LIN {X 0,Y 312.539,Z 409.82,A -85,B 0,C 180,E1 -15709.867,E2 -15709.867} C_VEL
LIN {X 0,Y 316.185,Z 420.984,A -85,B 0,C 180,E1 -15712.474,E2 -15712.474} C_VEL
LIN {X 0,Y 319.373,Z 431.927,A -85,B 0,C 180,E1 -15714.865,E2 -15714.865} C_VEL
LIN {X 0,Y 322.559,Z 445.519,A -85,B 0,C 180,E1 -15717.69,E2 -15717.69} C_VEL
LIN {X 0,Y 323.297,Z 449.924,A -85,B 0,C 180,E1 -15718.552,E2 -15718.552} C_VEL
LIN {X 0,Y 321.475,Z 469.515,A -85,B 0,C 180,E1 -15721.786,E2 -15721.786} C_VEL
LIN {X 0,Y 320.022,Z 488.05,A -85,B 0,C 180,E1 -15724.694,E2 -15724.694} C_VEL
LIN {X 0,Y 324.349,Z 518.766,A -85,B 0,C 180,E1 -15725.801,E2 -15725.801} C_VEL
LIN {X 0,Y 322.977,Z 585.301,A -85,B 0,C 180,E1 -15727.279,E2 -15727.279} C_VEL
LIN {X 0,Y 322.487,Z 602.467,A -85,B 0,C 180,E1 -15727.707,E2 -15727.707} C_VEL
LIN {X 0,Y 321.635,Z 615.557,A -85,B 0,C 180,E1 -15728.278,E2 -15728.278} C_VEL
LIN {X 0,Y 320.727,Z 627.617,A -85,B 0,C 180,E1 -15729.056,E2 -15729.056} C_VEL
LIN {X 0,Y 319.391,Z 639.348,A -85,B 0,C 180,E1 -15730.058,E2 -15730.058} C_VEL
LIN {X 0,Y 317.949,Z 650.541,A -85,B 0,C 180,E1 -15731.306,E2 -15731.306} C_VEL
LIN {X 0,Y 316.672,Z 660.214,A -85,B 0,C 180,E1 -15732.661,E2 -15732.661} C_VEL
LIN {X 0,Y 315.497,Z 668.968,A -85,B 0,C 180,E1 -15734.164,E2 -15734.164} C_VEL
LIN {X 0,Y 313.957,Z 677.978,A -85,B 0,C 180,E1 -15736.076,E2 -15736.076} C_VEL
LIN {X 0,Y 312.886,Z 685.206,A -85,B 0,C 180,E1 -15738.008,E2 -15738.008} C_VEL
LIN {X 0,Y 311.883,Z 691.838,A -85,B 0,C 180,E1 -15740.27,E2 -15740.27} C_VEL
LIN {X 0,Y 311.35,Z 696.194,A -85,B 0,C 180,E1 -15742.216,E2 -15742.216} C_VEL
LIN {X 0,Y 310.994,Z 699.108,A -85,B 0,C 180,E1 -15743.9,E2 -15743.9} C_VEL
LIN {X 0,Y 310.769,Z 701.783,A -85,B 0,C 180,E1 -15746.11,E2 -15746.11} C_VEL
LIN {X 0,Y 310.691,Z 702.783,A -85,B 0,C 180,E1 -15747.407,E2 -15747.407} C_VEL
LIN {X 0,Y 310.618,Z 703.635,A -85,B 0,C 180,E1 -15750,E2 -15750} C_VEL
LIN {X 0,Y 310.62,Z 703.44,A -85,B 0,C 180,E1 -15751.297,E2 -15751.297} C_VEL
LIN {X 0,Y 310.69,Z 702.849,A -85,B 0,C 180,E1 -15752.593,E2 -15752.593} C_VEL
LIN {X 0,Y 310.765,Z 701.874,A -85,B 0,C 180,E1 -15753.89,E2 -15753.89} C_VEL
LIN {X 0,Y 310.946,Z 699.383,A -85,B 0,C 180,E1 -15756.016,E2 -15756.016} C_VEL
LIN {X 0,Y 311.264,Z 696.397,A -85,B 0,C 180,E1 -15757.786,E2 -15757.786} C_VEL
LIN {X 0,Y 311.836,Z 692.102,A -85,B 0,C 180,E1 -15759.732,E2 -15759.732} C_VEL
LIN {X 0,Y 312.66,Z 686.615,A -85,B 0,C 180,E1 -15761.672,E2 -15761.672} C_VEL
LIN {X 0,Y 313.691,Z 679.736,A -85,B 0,C 180,E1 -15763.606,E2 -15763.606} C_VEL
LIN {X 0,Y 315.129,Z 671.132,A -85,B 0,C 180,E1 -15765.523,E2 -15765.523} C_VEL
LIN {X 0,Y 316.384,Z 662.938,A -85,B 0,C 180,E1 -15767.009,E2 -15767.009} C_VEL
LIN {X 0,Y 317.675,Z 652.616,A -85,B 0,C 180,E1 -15768.544,E2 -15768.544} C_VEL
LIN {X 0,Y 319.116,Z 641.878,A -85,B 0,C 180,E1 -15769.792,E2 -15769.792} C_VEL
LIN {X 0,Y 320.475,Z 629.948,A -85,B 0,C 180,E1 -15770.877,E2 -15770.877} C_VEL
LIN {X 0,Y 321.541,Z 617.429,A -85,B 0,C 180,E1 -15771.729,E2 -15771.729} C_VEL
LIN {X 0,Y 322.445,Z 604.145,A -85,B 0,C 180,E1 -15772.338,E2 -15772.338} C_VEL
LIN {X 0,Y 322.942,Z 589.97,A -85,B 0,C 180,E1 -15772.724,E2 -15772.724} C_VEL
LIN {X 0,Y 324.409,Z 518.731,A -85,B 0,C 180,E1 -15774.307,E2 -15774.307} C_VEL
LIN {X 0,Y 322.877,Z 507.001,A -85,B 0,C 180,E1 -15774.711,E2 -15774.711} C_VEL
LIN {X 0,Y 321.799,Z 503.315,A -85,B 0,C 180,E1 -15774.889,E2 -15774.889} C_VEL
LIN {X 0,Y 318.374,Z 497.993,A -85,B 0,C 180,E1 -15775.304,E2 -15775.304} C_VEL
LIN {X 0,Y 314.859,Z 492.705,A -85,B 0,C 180,E1 -15775.737,E2 -15775.737} C_VEL
LIN {X 0,Y 313.636,Z 489.058,A -85,B 0,C 180,E1 -15775.937,E2 -15775.937} C_VEL
LIN {X 0,Y 313.523,Z 487.144,A -85,B 0,C 180,E1 -15776.1,E2 -15776.1} C_VEL
LIN {X 0,Y 315.804,Z 461.684,A -85,B 0,C 180,E1 -15780.246,E2 -15780.246} C_VEL
LIN {X 0,Y 316.683,Z 451.244,A -85,B 0,C 180,E1 -15782.013,E2 -15782.013} C_VEL
LIN {X 0,Y 314.241,Z 439.793,A -85,B 0,C 180,E1 -15784.382,E2 -15784.382} C_VEL
LIN {X 0,Y 310.353,Z 425.27,A -85,B 0,C 180,E1 -15787.572,E2 -15787.572} C_VEL
LIN {X 0,Y 305.498,Z 410.99,A -85,B 0,C 180,E1 -15790.958,E2 -15790.958} C_VEL
LIN {X 0,Y 305.385,Z 410.45,A -85,B 0,C 180,E1 -15791.281,E2 -15791.281} C_VEL
LIN {X 0,Y 305.401,Z 410.414,A -85,B 0,C 180,E1 -15794.489,E2 -15794.489} C_VEL
LIN {X 0,Y 305.415,Z 410.443,A -85,B 0,C 180,E1 -15798.139,E2 -15798.139} C_VEL
LIN {X 0,Y 305.462,Z 410.432,A -85,B 0,C 180,E1 -15801.595,E2 -15801.595} C_VEL
LIN {X 0,Y 305.464,Z 410.436,A -85,B 0,C 180,E1 -15804.887,E2 -15804.887} C_VEL
LIN {X 0,Y 305.444,Z 410.439,A -85,B 0,C 180,E1 -15808.358,E2 -15808.358} C_VEL
LIN {X 0,Y 305.456,Z 410.422,A -85,B 0,C 180,E1 -15811.107,E2 -15811.107} C_VEL
LIN {X 0,Y 305.501,Z 410.431,A -85,B 0,C 180,E1 -15814.081,E2 -15814.081} C_VEL
LIN {X 0,Y 305.476,Z 410.417,A -85,B 0,C 180,E1 -15816.976,E2 -15816.976} C_VEL
LIN {X 0,Y 305.512,Z 410.414,A -85,B 0,C 180,E1 -15821.213,E2 -15821.213} C_VEL
LIN {X 0,Y 305.582,Z 410.421,A -85,B 0,C 180,E1 -15825.346,E2 -15825.346} C_VEL
LIN {X 0,Y 305.626,Z 410.392,A -85,B 0,C 180,E1 -15829.399,E2 -15829.399} C_VEL
LIN {X 0,Y 305.749,Z 410.399,A -85,B 0,C 180,E1 -15832.073,E2 -15832.073} C_VEL
LIN {X 0,Y 305.658,Z 410.387,A -85,B 0,C 180,E1 -15834.723,E2 -15834.723} C_VEL
LIN {X 0,Y 305.939,Z 410.374,A -85,B 0,C 180,E1 -15838.684,E2 -15838.684} C_VEL
LIN {X 0,Y 305.937,Z 410.356,A -85,B 0,C 180,E1 -15841.316,E2 -15841.316} C_VEL
LIN {X 0,Y 305.789,Z 410.393,A -85,B 0,C 180,E1 -15846.599,E2 -15846.599} C_VEL
LIN {X 0,Y 305.697,Z 410.381,A -85,B 0,C 180,E1 -15849.261,E2 -15849.261} C_VEL
LIN {X 0,Y 305.567,Z 410.422,A -85,B 0,C 180,E1 -15853.297,E2 -15853.297} C_VEL
LIN {X 0,Y 305.493,Z 410.407,A -85,B 0,C 180,E1 -15856.026,E2 -15856.026} C_VEL
LIN {X 0,Y 305.478,Z 410.433,A -85,B 0,C 180,E1 -15860.188,E2 -15860.188} C_VEL
LIN {X 0,Y 305.443,Z 410.425,A -85,B 0,C 180,E1 -15864.467,E2 -15864.467} C_VEL
LIN {X 0,Y 305.444,Z 410.431,A -85,B 0,C 180,E1 -15867.399,E2 -15867.399} C_VEL
LIN {X 0,Y 305.419,Z 410.43,A -85,B 0,C 180,E1 -15870.414,E2 -15870.414} C_VEL
LIN {X 0,Y 305.466,Z 410.419,A -85,B 0,C 180,E1 -15874.078,E2 -15874.078} C_VEL
LIN {X 0,Y 305.453,Z 410.437,A -85,B 0,C 180,E1 -15876.743,E2 -15876.743} C_VEL
LIN {X 0,Y 305.41,Z 410.388,A -85,B 0,C 180,E1 -15880.589,E2 -15880.589} C_VEL
LIN {X 0,Y 305.422,Z 410.412,A -85,B 0,C 180,E1 -15883.656,E2 -15883.656} C_VEL
LIN {X 0,Y 305.435,Z 410.407,A -85,B 0,C 180,E1 -15887.418,E2 -15887.418} C_VEL
LIN {X 0,Y 305.448,Z 410.435,A -85,B 0,C 180,E1 -15891.593,E2 -15891.593} C_VEL
LIN {X 0,Y 305.529,Z 410.634,A -85,B 0,C 180,E1 -15893.411,E2 -15893.411} C_VEL
LIN {X 0,Y 308.682,Z 425.243,A -85,B 0,C 180,E1 -15896.877,E2 -15896.877} C_VEL
LIN {X 0,Y 311.225,Z 437.046,A -85,B 0,C 180,E1 -15899.561,E2 -15899.561} C_VEL
LIN {X 0,Y 311.159,Z 440.07,A -85,B 0,C 180,E1 -15900.204,E2 -15900.204} C_VEL
LIN {X 0,Y 311.02,Z 441.837,A -85,B 0,C 180,E1 -15900.497,E2 -15900.497} C_VEL
LIN {X 0,Y 312.83,Z 473.685,A -85,B 0,C 180,E1 -15903.011,E2 -15903.011} C_VEL
LIN {X 0,Y 313.362,Z 488.832,A -85,B 0,C 180,E1 -15904.212,E2 -15904.212} C_VEL
LIN {X 0,Y 316.809,Z 520.766,A -85,B 0,C 180,E1 -15905.295,E2 -15905.295} C_VEL
LIN {X 0,Y 317.335,Z 528.316,A -85,B 0,C 180,E1 -15905.522,E2 -15905.522} C_VEL
LIN {X 0,Y 315.578,Z 604.063,A -85,B 0,C 180,E1 -15907.235,E2 -15907.235} C_VEL
LIN {X 0,Y 314.795,Z 617.344,A -85,B 0,C 180,E1 -15907.738,E2 -15907.738} C_VEL
LIN {X 0,Y 313.773,Z 629.822,A -85,B 0,C 180,E1 -15908.483,E2 -15908.483} C_VEL
LIN {X 0,Y 312.624,Z 641.462,A -85,B 0,C 180,E1 -15909.435,E2 -15909.435} C_VEL
LIN {X 0,Y 311.242,Z 652.056,A -85,B 0,C 180,E1 -15910.545,E2 -15910.545} C_VEL
LIN {X 0,Y 309.74,Z 662.85,A -85,B 0,C 180,E1 -15911.992,E2 -15911.992} C_VEL
LIN {X 0,Y 308.35,Z 672.278,A -85,B 0,C 180,E1 -15913.57,E2 -15913.57} C_VEL
LIN {X 0,Y 307.006,Z 681.154,A -85,B 0,C 180,E1 -15915.415,E2 -15915.415} C_VEL
LIN {X 0,Y 305.735,Z 688.702,A -85,B 0,C 180,E1 -15917.386,E2 -15917.386} C_VEL
LIN {X 0,Y 304.903,Z 694.761,A -85,B 0,C 180,E1 -15919.374,E2 -15919.374} C_VEL
LIN {X 0,Y 304.256,Z 699.543,A -85,B 0,C 180,E1 -15921.365,E2 -15921.365} C_VEL
LIN {X 0,Y 303.913,Z 703.193,A -85,B 0,C 180,E1 -15923.36,E2 -15923.36} C_VEL
LIN {X 0,Y 303.761,Z 705.073,A -85,B 0,C 180,E1 -15924.69,E2 -15924.69} C_VEL
LIN {X 0,Y 303.702,Z 706.49,A -85,B 0,C 180,E1 -15926.019,E2 -15926.019} C_VEL
LIN {X 0,Y 303.658,Z 707.49,A -85,B 0,C 180,E1 -15927.347,E2 -15927.347} C_VEL
LIN {X 0,Y 303.597,Z 708.1,A -85,B 0,C 180,E1 -15928.673,E2 -15928.673} C_VEL
LIN {X 0,Y 303.616,Z 708.317,A -85,B 0,C 180,E1 -15930,E2 -15930} C_VEL
LIN {X 0,Y 303.626,Z 708.094,A -85,B 0,C 180,E1 -15931.326,E2 -15931.326} C_VEL
LIN {X 0,Y 303.665,Z 707.479,A -85,B 0,C 180,E1 -15932.653,E2 -15932.653} C_VEL
LIN {X 0,Y 303.723,Z 706.475,A -85,B 0,C 180,E1 -15933.98,E2 -15933.98} C_VEL
LIN {X 0,Y 303.825,Z 704.233,A -85,B 0,C 180,E1 -15935.92,E2 -15935.92} C_VEL
LIN {X 0,Y 304.103,Z 700.848,A -85,B 0,C 180,E1 -15937.97,E2 -15937.97} C_VEL
LIN {X 0,Y 304.692,Z 696.451,A -85,B 0,C 180,E1 -15939.962,E2 -15939.962} C_VEL
LIN {X 0,Y 305.604,Z 689.751,A -85,B 0,C 180,E1 -15942.282,E2 -15942.282} C_VEL
LIN {X 0,Y 306.777,Z 682.429,A -85,B 0,C 180,E1 -15944.257,E2 -15944.257} C_VEL
LIN {X 0,Y 308.121,Z 673.606,A -85,B 0,C 180,E1 -15946.163,E2 -15946.163} C_VEL
LIN {X 0,Y 309.554,Z 663.768,A -85,B 0,C 180,E1 -15947.848,E2 -15947.848} C_VEL
LIN {X 0,Y 311.059,Z 653.202,A -85,B 0,C 180,E1 -15949.295,E2 -15949.295} C_VEL
LIN {X 0,Y 312.382,Z 642.956,A -85,B 0,C 180,E1 -15950.409,E2 -15950.409} C_VEL
LIN {X 0,Y 313.685,Z 630.643,A -85,B 0,C 180,E1 -15951.437,E2 -15951.437} C_VEL
LIN {X 0,Y 314.762,Z 618.361,A -85,B 0,C 180,E1 -15952.221,E2 -15952.221} C_VEL
LIN {X 0,Y 317.898,Z 604.839,A -85,B 0,C 180,E1 -15953.622,E2 -15953.622} C_VEL
LIN {X 0,Y 320.563,Z 591.482,A -85,B 0,C 180,E1 -15954.704,E2 -15954.704} C_VEL
LIN {X 0,Y 322.77,Z 577.813,A -85,B 0,C 180,E1 -15955.556,E2 -15955.556} C_VEL
LIN {X 0,Y 324.493,Z 563.284,A -85,B 0,C 180,E1 -15956.229,E2 -15956.229} C_VEL
LIN {X 0,Y 327.437,Z 528.631,A -85,B 0,C 180,E1 -15957.532,E2 -15957.532} C_VEL
LIN {X 0,Y 327.503,Z 512.069,A -85,B 0,C 180,E1 -15958.423,E2 -15958.423} C_VEL
LIN {X 0,Y 326.752,Z 496.351,A -85,B 0,C 180,E1 -15959.479,E2 -15959.479} C_VEL
LIN {X 0,Y 325.256,Z 480.762,A -85,B 0,C 180,E1 -15960.768,E2 -15960.768} C_VEL
LIN {X 0,Y 323.384,Z 466.341,A -85,B 0,C 180,E1 -15962.201,E2 -15962.201} C_VEL
LIN {X 0,Y 322.036,Z 457.299,A -85,B 0,C 180,E1 -15963.249,E2 -15963.249} C_VEL
LIN {X 0,Y 319.695,Z 451.276,A -85,B 0,C 180,E1 -15964.432,E2 -15964.432} C_VEL
LIN {X 0,Y 315.876,Z 442.522,A -85,B 0,C 180,E1 -15966.702,E2 -15966.702} C_VEL
LIN {X 0,Y 314.394,Z 436.999,A -85,B 0,C 180,E1 -15969.172,E2 -15969.172} C_VEL
LIN {X 0,Y 313.453,Z 433.635,A -85,B 0,C 180,E1 -15970.993,E2 -15970.993} C_VEL
LIN {X 0,Y 312.007,Z 429.364,A -85,B 0,C 180,E1 -15973.879,E2 -15973.879} C_VEL
LIN {X 0,Y 310.757,Z 425.66,A -85,B 0,C 180,E1 -15977.276,E2 -15977.276} C_VEL
LIN {X 0,Y 310.242,Z 424.091,A -85,B 0,C 180,E1 -15979.629,E2 -15979.629} C_VEL
LIN {X 0,Y 311.764,Z 424.945,A -85,B 0,C 180,E1 -15981.669,E2 -15981.669} C_VEL
LIN {X 0,Y 313.944,Z 425.846,A -85,B 0,C 180,E1 -15983.379,E2 -15983.379} C_VEL
LIN {X 0,Y 316.792,Z 428.045,A -85,B 0,C 180,E1 -15985.169,E2 -15985.169} C_VEL
LIN {X 0,Y 320.809,Z 431.911,A -85,B 0,C 180,E1 -15987.214,E2 -15987.214} C_VEL
LIN {X 0,Y 323.364,Z 434.77,A -85,B 0,C 180,E1 -15988.331,E2 -15988.331} C_VEL
LIN {X 0,Y 324.917,Z 437.076,A -85,B 0,C 180,E1 -15989,E2 -15989} C_VEL
LIN {X 0,Y 329.004,Z 443.809,A -85,B 0,C 180,E1 -15990.619,E2 -15990.619} C_VEL
LIN {X 0,Y 333.23,Z 452.024,A -85,B 0,C 180,E1 -15992.145,E2 -15992.145} C_VEL
LIN {X 0,Y 329.446,Z 489.733,A -85,B 0,C 180,E1 -15993.634,E2 -15993.634} C_VEL
LIN {X 0,Y 328.128,Z 509.636,A -85,B 0,C 180,E1 -15994.552,E2 -15994.552} C_VEL
LIN {X 0,Y 326.845,Z 523.763,A -85,B 0,C 180,E1 -15995.472,E2 -15995.472} C_VEL
LIN {X 0,Y 325.453,Z 535.265,A -85,B 0,C 180,E1 -15996.453,E2 -15996.453} C_VEL
LIN {X 0,Y 323.679,Z 546.599,A -85,B 0,C 180,E1 -15997.668,E2 -15997.668} C_VEL
LIN {X 0,Y 321.413,Z 557.833,A -85,B 0,C 180,E1 -15999.187,E2 -15999.187} C_VEL
LIN {X 0,Y 319.436,Z 566.96,A -85,B 0,C 180,E1 -16000.73,E2 -16000.73} C_VEL
LIN {X 0,Y 317.213,Z 575.546,A -85,B 0,C 180,E1 -16002.534,E2 -16002.534} C_VEL
LIN {X 0,Y 315.008,Z 582.876,A -85,B 0,C 180,E1 -16004.471,E2 -16004.471} C_VEL
LIN {X 0,Y 313.158,Z 588.479,A -85,B 0,C 180,E1 -16006.37,E2 -16006.37} C_VEL
LIN {X 0,Y 311.44,Z 592.85,A -85,B 0,C 180,E1 -16008.282,E2 -16008.282} C_VEL
LIN {X 0,Y 310.478,Z 595.11,A -85,B 0,C 180,E1 -16009.567,E2 -16009.567} C_VEL
LIN {X 0,Y 309.561,Z 596.914,A -85,B 0,C 180,E1 -16010.856,E2 -16010.856} C_VEL
LIN {X 0,Y 308.695,Z 598.235,A -85,B 0,C 180,E1 -16012.149,E2 -16012.149} C_VEL
LIN {X 0,Y 308.072,Z 599.122,A -85,B 0,C 180,E1 -16013.45,E2 -16013.45} C_VEL
LIN {X 0,Y 307.598,Z 599.575,A -85,B 0,C 180,E1 -16014.756,E2 -16014.756} C_VEL
LIN {X 0,Y 307.124,Z 599.575,A -85,B 0,C 180,E1 -16016.064,E2 -16016.064} C_VEL
LIN {X 0,Y 306.617,Z 599.175,A -85,B 0,C 180,E1 -16017.373,E2 -16017.373} C_VEL
LIN {X 0,Y 306.293,Z 598.342,A -85,B 0,C 180,E1 -16018.685,E2 -16018.685} C_VEL
LIN {X 0,Y 305.867,Z 597.074,A -85,B 0,C 180,E1 -16020,E2 -16020} C_VEL
LIN {X 0,Y 305.752,Z 594.31,A -85,B 0,C 180,E1 -16021.976,E2 -16021.976} C_VEL
LIN {X 0,Y 305.613,Z 590.502,A -85,B 0,C 180,E1 -16023.956,E2 -16023.956} C_VEL
LIN {X 0,Y 305.81,Z 585.528,A -85,B 0,C 180,E1 -16025.936,E2 -16025.936} C_VEL
LIN {X 0,Y 306.111,Z 579.272,A -85,B 0,C 180,E1 -16027.918,E2 -16027.918} C_VEL
LIN {X 0,Y 306.582,Z 571.477,A -85,B 0,C 180,E1 -16029.914,E2 -16029.914} C_VEL
LIN {X 0,Y 307.077,Z 561.898,A -85,B 0,C 180,E1 -16031.887,E2 -16031.887} C_VEL
LIN {X 0,Y 307.669,Z 552.084,A -85,B 0,C 180,E1 -16033.541,E2 -16033.541} C_VEL
LIN {X 0,Y 308.288,Z 541.233,A -85,B 0,C 180,E1 -16035.029,E2 -16035.029} C_VEL
LIN {X 0,Y 308.947,Z 529.369,A -85,B 0,C 180,E1 -16036.35,E2 -16036.35} C_VEL
LIN {X 0,Y 309.453,Z 516.504,A -85,B 0,C 180,E1 -16037.471,E2 -16037.471} C_VEL
LIN {X 0,Y 309.903,Z 503.178,A -85,B 0,C 180,E1 -16038.352,E2 -16038.352} C_VEL
LIN {X 0,Y 310.218,Z 488.806,A -85,B 0,C 180,E1 -16039.006,E2 -16039.006} C_VEL
LIN {X 0,Y 311.04,Z 448.886,A -85,B 0,C 180,E1 -16040.32,E2 -16040.32} C_VEL
LIN {X 0,Y 311.496,Z 430.443,A -85,B 0,C 180,E1 -16040.934,E2 -16040.934} C_VEL
LIN {X 0,Y 305.728,Z 411.446,A -85,B 0,C 180,E1 -16041.846,E2 -16041.846} C_VEL
LIN {X 0,Y 305.565,Z 410.535,A -85,B 0,C 180,E1 -16042.08,E2 -16042.08} C_VEL
LIN {X 0,Y 305.475,Z 410.434,A -85,B 0,C 180,E1 -16046.199,E2 -16046.199} C_VEL
LIN {X 0,Y 305.46,Z 410.416,A -85,B 0,C 180,E1 -16049.037,E2 -16049.037} C_VEL
LIN {X 0,Y 305.438,Z 410.439,A -85,B 0,C 180,E1 -16051.953,E2 -16051.953} C_VEL
LIN {X 0,Y 305.464,Z 410.426,A -85,B 0,C 180,E1 -16055.113,E2 -16055.113} C_VEL
LIN {X 0,Y 305.442,Z 410.426,A -85,B 0,C 180,E1 -16058.527,E2 -16058.527} C_VEL
LIN {X 0,Y 305.456,Z 410.428,A -85,B 0,C 180,E1 -16062.586,E2 -16062.586} C_VEL
LIN {X 0,Y 305.427,Z 410.438,A -85,B 0,C 180,E1 -16066.345,E2 -16066.345} C_VEL
LIN {X 0,Y 305.476,Z 410.634,A -85,B 0,C 180,E1 -16069.052,E2 -16069.052} C_VEL
LIN {X 0,Y 309.593,Z 423.12,A -85,B 0,C 180,E1 -16072.086,E2 -16072.086} C_VEL
LIN {X 0,Y 312.806,Z 434.138,A -85,B 0,C 180,E1 -16074.532,E2 -16074.532} C_VEL
LIN {X 0,Y 316.219,Z 448.825,A -85,B 0,C 180,E1 -16077.625,E2 -16077.625} C_VEL
LIN {X 0,Y 316.664,Z 452.335,A -85,B 0,C 180,E1 -16078.302,E2 -16078.302} C_VEL
LIN {X 0,Y 314.685,Z 472.51,A -85,B 0,C 180,E1 -16081.668,E2 -16081.668} C_VEL
LIN {X 0,Y 313.435,Z 487.99,A -85,B 0,C 180,E1 -16084.12,E2 -16084.12} C_VEL
LIN {X 0,Y 317.883,Z 519.622,A -85,B 0,C 180,E1 -16085.298,E2 -16085.298} C_VEL
LIN {X 0,Y 316.456,Z 585.266,A -85,B 0,C 180,E1 -16086.784,E2 -16086.784} C_VEL
LIN {X 0,Y 315.946,Z 602.471,A -85,B 0,C 180,E1 -16087.22,E2 -16087.22} C_VEL
LIN {X 0,Y 315.06,Z 615.582,A -85,B 0,C 180,E1 -16087.801,E2 -16087.801} C_VEL
LIN {X 0,Y 314.116,Z 627.654,A -85,B 0,C 180,E1 -16088.594,E2 -16088.594} C_VEL
LIN {X 0,Y 312.737,Z 639.391,A -85,B 0,C 180,E1 -16089.615,E2 -16089.615} C_VEL
LIN {X 0,Y 311.233,Z 650.587,A -85,B 0,C 180,E1 -16090.887,E2 -16090.887} C_VEL
LIN {X 0,Y 309.698,Z 661.567,A -85,B 0,C 180,E1 -16092.473,E2 -16092.473} C_VEL
LIN {X 0,Y 308.342,Z 670.653,A -85,B 0,C 180,E1 -16094.127,E2 -16094.127} C_VEL
LIN {X 0,Y 306.834,Z 679.356,A -85,B 0,C 180,E1 -16096.084,E2 -16096.084} C_VEL
LIN {X 0,Y 305.743,Z 686.341,A -85,B 0,C 180,E1 -16098.061,E2 -16098.061} C_VEL
LIN {X 0,Y 304.861,Z 691.892,A -85,B 0,C 180,E1 -16100.044,E2 -16100.044} C_VEL
LIN {X 0,Y 304.294,Z 696.248,A -85,B 0,C 180,E1 -16102.035,E2 -16102.035} C_VEL
LIN {X 0,Y 303.886,Z 699.461,A -85,B 0,C 180,E1 -16103.971,E2 -16103.971} C_VEL
LIN {X 0,Y 303.687,Z 701.837,A -85,B 0,C 180,E1 -16106.019,E2 -16106.019} C_VEL
LIN {X 0,Y 303.617,Z 702.837,A -85,B 0,C 180,E1 -16107.347,E2 -16107.347} C_VEL
LIN {X 0,Y 303.535,Z 703.689,A -85,B 0,C 180,E1 -16110,E2 -16110} C_VEL
LIN {X 0,Y 303.539,Z 703.493,A -85,B 0,C 180,E1 -16111.327,E2 -16111.327} C_VEL
LIN {X 0,Y 303.617,Z 702.902,A -85,B 0,C 180,E1 -16112.654,E2 -16112.654} C_VEL
LIN {X 0,Y 303.683,Z 701.928,A -85,B 0,C 180,E1 -16113.981,E2 -16113.981} C_VEL
LIN {X 0,Y 303.872,Z 699.638,A -85,B 0,C 180,E1 -16116.004,E2 -16116.004} C_VEL
LIN {X 0,Y 304.231,Z 696.449,A -85,B 0,C 180,E1 -16117.967,E2 -16117.967} C_VEL
LIN {X 0,Y 304.817,Z 692.153,A -85,B 0,C 180,E1 -16119.958,E2 -16119.958} C_VEL
LIN {X 0,Y 305.694,Z 686.665,A -85,B 0,C 180,E1 -16121.942,E2 -16121.942} C_VEL
LIN {X 0,Y 306.78,Z 679.784,A -85,B 0,C 180,E1 -16123.919,E2 -16123.919} C_VEL
LIN {X 0,Y 308.281,Z 671.178,A -85,B 0,C 180,E1 -16125.877,E2 -16125.877} C_VEL
LIN {X 0,Y 309.668,Z 661.826,A -85,B 0,C 180,E1 -16127.597,E2 -16127.597} C_VEL
LIN {X 0,Y 311.131,Z 651.407,A -85,B 0,C 180,E1 -16129.119,E2 -16129.119} C_VEL
LIN {X 0,Y 312.649,Z 640.386,A -85,B 0,C 180,E1 -16130.391,E2 -16130.391} C_VEL
LIN {X 0,Y 313.853,Z 629.974,A -85,B 0,C 180,E1 -16131.339,E2 -16131.339} C_VEL
LIN {X 0,Y 314.972,Z 617.437,A -85,B 0,C 180,E1 -16132.206,E2 -16132.206} C_VEL
LIN {X 0,Y 315.899,Z 604.125,A -85,B 0,C 180,E1 -16132.827,E2 -16132.827} C_VEL
LIN {X 0,Y 316.419,Z 589.888,A -85,B 0,C 180,E1 -16133.219,E2 -16133.219} C_VEL
LIN {X 0,Y 317.94,Z 519.507,A -85,B 0,C 180,E1 -16134.813,E2 -16134.813} C_VEL
LIN {X 0,Y 313.636,Z 489.058,A -85,B 0,C 180,E1 -16135.937,E2 -16135.937} C_VEL
LIN {X 0,Y 312.94,Z 486.827,A -85,B 0,C 180,E1 -16136.204,E2 -16136.204} C_VEL
LIN {X 0,Y 310.285,Z 479.752,A -85,B 0,C 180,E1 -16137.628,E2 -16137.628} C_VEL
LIN {X 0,Y 308.746,Z 472.042,A -85,B 0,C 180,E1 -16139.145,E2 -16139.145} C_VEL
LIN {X 0,Y 308.815,Z 467.004,A -85,B 0,C 180,E1 -16140.001,E2 -16140.001} C_VEL
LIN {X 0,Y 310.097,Z 454.673,A -85,B 0,C 180,E1 -16142.095,E2 -16142.095} C_VEL
LIN {X 0,Y 309.637,Z 450.645,A -85,B 0,C 180,E1 -16142.88,E2 -16142.88} C_VEL
LIN {X 0,Y 306.672,Z 438.007,A -85,B 0,C 180,E1 -16145.596,E2 -16145.596} C_VEL
LIN {X 0,Y 303.141,Z 425.405,A -85,B 0,C 180,E1 -16148.467,E2 -16148.467} C_VEL
LIN {X 0,Y 298.41,Z 411.555,A -85,B 0,C 180,E1 -16151.906,E2 -16151.906} C_VEL
LIN {X 0,Y 298.373,Z 411.305,A -85,B 0,C 180,E1 -16153.098,E2 -16153.098} C_VEL
LIN {X 0,Y 298.373,Z 411.313,A -85,B 0,C 180,E1 -16156.915,E2 -16156.915} C_VEL
LIN {X 0,Y 298.387,Z 411.32,A -85,B 0,C 180,E1 -16161.011,E2 -16161.011} C_VEL
LIN {X 0,Y 298.407,Z 411.311,A -85,B 0,C 180,E1 -16163.928,E2 -16163.928} C_VEL
LIN {X 0,Y 298.395,Z 411.303,A -85,B 0,C 180,E1 -16167.2,E2 -16167.2} C_VEL
LIN {X 0,Y 298.367,Z 411.306,A -85,B 0,C 180,E1 -16170.638,E2 -16170.638} C_VEL
LIN {X 0,Y 298.441,Z 411.304,A -85,B 0,C 180,E1 -16174.92,E2 -16174.92} C_VEL
LIN {X 0,Y 298.402,Z 411.306,A -85,B 0,C 180,E1 -16177.862,E2 -16177.862} C_VEL
LIN {X 0,Y 298.463,Z 411.298,A -85,B 0,C 180,E1 -16180.752,E2 -16180.752} C_VEL
LIN {X 0,Y 298.514,Z 411.3,A -85,B 0,C 180,E1 -16184.991,E2 -16184.991} C_VEL
LIN {X 0,Y 298.584,Z 411.267,A -85,B 0,C 180,E1 -16189.146,E2 -16189.146} C_VEL
LIN {X 0,Y 298.701,Z 411.279,A -85,B 0,C 180,E1 -16191.884,E2 -16191.884} C_VEL
LIN {X 0,Y 298.628,Z 411.263,A -85,B 0,C 180,E1 -16194.598,E2 -16194.598} C_VEL
LIN {X 0,Y 298.907,Z 411.25,A -85,B 0,C 180,E1 -16198.653,E2 -16198.653} C_VEL
LIN {X 0,Y 298.905,Z 411.23,A -85,B 0,C 180,E1 -16201.347,E2 -16201.347} C_VEL
LIN {X 0,Y 298.738,Z 411.271,A -85,B 0,C 180,E1 -16206.755,E2 -16206.755} C_VEL
LIN {X 0,Y 298.628,Z 411.26,A -85,B 0,C 180,E1 -16209.482,E2 -16209.482} C_VEL
LIN {X 0,Y 298.518,Z 411.301,A -85,B 0,C 180,E1 -16213.617,E2 -16213.617} C_VEL
LIN {X 0,Y 298.43,Z 411.284,A -85,B 0,C 180,E1 -16216.415,E2 -16216.415} C_VEL
LIN {X 0,Y 298.433,Z 411.311,A -85,B 0,C 180,E1 -16219.611,E2 -16219.611} C_VEL
LIN {X 0,Y 298.384,Z 411.294,A -85,B 0,C 180,E1 -16223.604,E2 -16223.604} C_VEL
LIN {X 0,Y 298.403,Z 411.313,A -85,B 0,C 180,E1 -16226.583,E2 -16226.583} C_VEL
LIN {X 0,Y 298.359,Z 411.301,A -85,B 0,C 180,E1 -16229.648,E2 -16229.648} C_VEL
LIN {X 0,Y 298.395,Z 411.313,A -85,B 0,C 180,E1 -16232.8,E2 -16232.8} C_VEL
LIN {X 0,Y 298.405,Z 411.31,A -85,B 0,C 180,E1 -16236.072,E2 -16236.072} C_VEL
LIN {X 0,Y 298.375,Z 411.279,A -85,B 0,C 180,E1 -16239.492,E2 -16239.492} C_VEL
LIN {X 0,Y 298.37,Z 411.276,A -85,B 0,C 180,E1 -16243.097,E2 -16243.097} C_VEL
LIN {X 0,Y 298.371,Z 411.296,A -85,B 0,C 180,E1 -16246.914,E2 -16246.914} C_VEL
LIN {X 0,Y 298.356,Z 411.301,A -85,B 0,C 180,E1 -16251.018,E2 -16251.018} C_VEL
LIN {X 0,Y 298.497,Z 411.542,A -85,B 0,C 180,E1 -16253.18,E2 -16253.18} C_VEL
LIN {X 0,Y 301.836,Z 427.164,A -85,B 0,C 180,E1 -16256.954,E2 -16256.954} C_VEL
LIN {X 0,Y 304.14,Z 437.746,A -85,B 0,C 180,E1 -16259.365,E2 -16259.365} C_VEL
LIN {X 0,Y 304.859,Z 443.301,A -85,B 0,C 180,E1 -16259.907,E2 -16259.907} C_VEL
LIN {X 0,Y 306.463,Z 474.151,A -85,B 0,C 180,E1 -16262.416,E2 -16262.416} C_VEL
LIN {X 0,Y 306.86,Z 488.84,A -85,B 0,C 180,E1 -16263.622,E2 -16263.622} C_VEL
LIN {X 0,Y 310.309,Z 520.688,A -85,B 0,C 180,E1 -16264.738,E2 -16264.738} C_VEL
LIN {X 0,Y 310.859,Z 529.725,A -85,B 0,C 180,E1 -16265.01,E2 -16265.01} C_VEL
LIN {X 0,Y 309.063,Z 604.111,A -85,B 0,C 180,E1 -16266.727,E2 -16266.727} C_VEL
LIN {X 0,Y 308.275,Z 616.535,A -85,B 0,C 180,E1 -16267.197,E2 -16267.197} C_VEL
LIN {X 0,Y 307.286,Z 628.691,A -85,B 0,C 180,E1 -16267.917,E2 -16267.917} C_VEL
LIN {X 0,Y 305.995,Z 641.431,A -85,B 0,C 180,E1 -16268.969,E2 -16268.969} C_VEL
LIN {X 0,Y 304.567,Z 652.019,A -85,B 0,C 180,E1 -16270.101,E2 -16270.101} C_VEL
LIN {X 0,Y 302.967,Z 662.807,A -85,B 0,C 180,E1 -16271.575,E2 -16271.575} C_VEL
LIN {X 0,Y 301.485,Z 672.554,A -85,B 0,C 180,E1 -16273.249,E2 -16273.249} C_VEL
LIN {X 0,Y 300.133,Z 681.106,A -85,B 0,C 180,E1 -16275.073,E2 -16275.073} C_VEL
LIN {X 0,Y 298.794,Z 688.652,A -85,B 0,C 180,E1 -16277.088,E2 -16277.088} C_VEL
LIN {X 0,Y 297.885,Z 694.71,A -85,B 0,C 180,E1 -16279.12,E2 -16279.12} C_VEL
LIN {X 0,Y 297.217,Z 699.491,A -85,B 0,C 180,E1 -16281.158,E2 -16281.158} C_VEL
LIN {X 0,Y 296.846,Z 703.14,A -85,B 0,C 180,E1 -16283.201,E2 -16283.201} C_VEL
LIN {X 0,Y 296.689,Z 705.02,A -85,B 0,C 180,E1 -16284.563,E2 -16284.563} C_VEL
LIN {X 0,Y 296.601,Z 706.437,A -85,B 0,C 180,E1 -16285.923,E2 -16285.923} C_VEL
LIN {X 0,Y 296.584,Z 707.437,A -85,B 0,C 180,E1 -16287.283,E2 -16287.283} C_VEL
LIN {X 0,Y 296.516,Z 708.047,A -85,B 0,C 180,E1 -16288.642,E2 -16288.642} C_VEL
LIN {X 0,Y 296.53,Z 708.263,A -85,B 0,C 180,E1 -16290,E2 -16290} C_VEL
LIN {X 0,Y 296.544,Z 708.04,A -85,B 0,C 180,E1 -16291.358,E2 -16291.358} C_VEL
LIN {X 0,Y 296.59,Z 707.425,A -85,B 0,C 180,E1 -16292.716,E2 -16292.716} C_VEL
LIN {X 0,Y 296.639,Z 706.421,A -85,B 0,C 180,E1 -16294.076,E2 -16294.076} C_VEL
LIN {X 0,Y 296.738,Z 704.415,A -85,B 0,C 180,E1 -16295.88,E2 -16295.88} C_VEL
LIN {X 0,Y 297.061,Z 700.794,A -85,B 0,C 180,E1 -16298.161,E2 -16298.161} C_VEL
LIN {X 0,Y 297.66,Z 696.397,A -85,B 0,C 180,E1 -16300.2,E2 -16300.2} C_VEL
LIN {X 0,Y 298.625,Z 689.697,A -85,B 0,C 180,E1 -16302.574,E2 -16302.574} C_VEL
LIN {X 0,Y 299.869,Z 682.377,A -85,B 0,C 180,E1 -16304.593,E2 -16304.593} C_VEL
LIN {X 0,Y 301.266,Z 673.71,A -85,B 0,C 180,E1 -16306.51,E2 -16306.51} C_VEL
LIN {X 0,Y 302.792,Z 663.719,A -85,B 0,C 180,E1 -16308.261,E2 -16308.261} C_VEL
LIN {X 0,Y 304.375,Z 653.156,A -85,B 0,C 180,E1 -16309.736,E2 -16309.736} C_VEL
LIN {X 0,Y 305.728,Z 642.914,A -85,B 0,C 180,E1 -16310.874,E2 -16310.874} C_VEL
LIN {X 0,Y 307.095,Z 630.609,A -85,B 0,C 180,E1 -16311.92,E2 -16311.92} C_VEL
LIN {X 0,Y 307.982,Z 620.933,A -85,B 0,C 180,E1 -16312.56,E2 -16312.56} C_VEL
LIN {X 0,Y 311.125,Z 608.476,A -85,B 0,C 180,E1 -16313.991,E2 -16313.991} C_VEL
LIN {X 0,Y 314.052,Z 595.572,A -85,B 0,C 180,E1 -16315.163,E2 -16315.163} C_VEL
LIN {X 0,Y 316.719,Z 581.3,A -85,B 0,C 180,E1 -16316.169,E2 -16316.169} C_VEL
LIN {X 0,Y 318.938,Z 566.333,A -85,B 0,C 180,E1 -16316.943,E2 -16316.943} C_VEL
LIN {X 0,Y 322.373,Z 529.81,A -85,B 0,C 180,E1 -16318.378,E2 -16318.378} C_VEL
LIN {X 0,Y 322.579,Z 513.411,A -85,B 0,C 180,E1 -16319.298,E2 -16319.298} C_VEL
LIN {X 0,Y 322.034,Z 498.47,A -85,B 0,C 180,E1 -16320.345,E2 -16320.345} C_VEL
LIN {X 0,Y 320.86,Z 483.7,A -85,B 0,C 180,E1 -16321.608,E2 -16321.608} C_VEL
LIN {X 0,Y 319.33,Z 469.773,A -85,B 0,C 180,E1 -16323.037,E2 -16323.037} C_VEL
LIN {X 0,Y 318.265,Z 461.755,A -85,B 0,C 180,E1 -16323.994,E2 -16323.994} C_VEL
LIN {X 0,Y 316.441,Z 456.645,A -85,B 0,C 180,E1 -16325.045,E2 -16325.045} C_VEL
LIN {X 0,Y 312.699,Z 447.681,A -85,B 0,C 180,E1 -16327.447,E2 -16327.447} C_VEL
LIN {X 0,Y 309.214,Z 440.368,A -85,B 0,C 180,E1 -16330.353,E2 -16330.353} C_VEL
LIN {X 0,Y 307.507,Z 435.89,A -85,B 0,C 180,E1 -16332.862,E2 -16332.862} C_VEL
LIN {X 0,Y 306.833,Z 433.197,A -85,B 0,C 180,E1 -16335.239,E2 -16335.239} C_VEL
LIN {X 0,Y 307.058,Z 431.726,A -85,B 0,C 180,E1 -16337.332,E2 -16337.332} C_VEL
LIN {X 0,Y 307.757,Z 431.059,A -85,B 0,C 180,E1 -16338.903,E2 -16338.903} C_VEL
LIN {X 0,Y 309.708,Z 431.684,A -85,B 0,C 180,E1 -16341.415,E2 -16341.415} C_VEL
LIN {X 0,Y 311.962,Z 432.588,A -85,B 0,C 180,E1 -16343.231,E2 -16343.231} C_VEL
LIN {X 0,Y 314.638,Z 434.745,A -85,B 0,C 180,E1 -16344.971,E2 -16344.971} C_VEL
LIN {X 0,Y 318.216,Z 438.206,A -85,B 0,C 180,E1 -16346.865,E2 -16346.865} C_VEL
LIN {X 0,Y 320.775,Z 441.286,A -85,B 0,C 180,E1 -16348.069,E2 -16348.069} C_VEL
LIN {X 0,Y 323.58,Z 445.937,A -85,B 0,C 180,E1 -16349.332,E2 -16349.332} C_VEL
LIN {X 0,Y 327.171,Z 452.586,A -85,B 0,C 180,E1 -16350.785,E2 -16350.785} C_VEL
LIN {X 0,Y 328.486,Z 455.414,A -85,B 0,C 180,E1 -16351.307,E2 -16351.307} C_VEL
LIN {X 0,Y 324.625,Z 491.379,A -85,B 0,C 180,E1 -16352.765,E2 -16352.765} C_VEL
LIN {X 0,Y 323.109,Z 511.39,A -85,B 0,C 180,E1 -16353.724,E2 -16353.724} C_VEL
LIN {X 0,Y 321.841,Z 524.554,A -85,B 0,C 180,E1 -16354.587,E2 -16354.587} C_VEL
LIN {X 0,Y 320.358,Z 535.61,A -85,B 0,C 180,E1 -16355.539,E2 -16355.539} C_VEL
LIN {X 0,Y 318.194,Z 548.239,A -85,B 0,C 180,E1 -16356.918,E2 -16356.918} C_VEL
LIN {X 0,Y 315.813,Z 559.447,A -85,B 0,C 180,E1 -16358.458,E2 -16358.458} C_VEL
LIN {X 0,Y 313.677,Z 568.428,A -85,B 0,C 180,E1 -16360.021,E2 -16360.021} C_VEL
LIN {X 0,Y 311.012,Z 577.825,A -85,B 0,C 180,E1 -16362.066,E2 -16362.066} C_VEL
LIN {X 0,Y 308.533,Z 585.266,A -85,B 0,C 180,E1 -16364.137,E2 -16364.137} C_VEL
LIN {X 0,Y 306.568,Z 590.595,A -85,B 0,C 180,E1 -16366.072,E2 -16366.072} C_VEL
LIN {X 0,Y 304.745,Z 594.739,A -85,B 0,C 180,E1 -16368.021,E2 -16368.021} C_VEL
LIN {X 0,Y 303.721,Z 596.897,A -85,B 0,C 180,E1 -16369.332,E2 -16369.332} C_VEL
LIN {X 0,Y 302.747,Z 598.549,A -85,B 0,C 180,E1 -16370.648,E2 -16370.648} C_VEL
LIN {X 0,Y 301.841,Z 599.774,A -85,B 0,C 180,E1 -16371.969,E2 -16371.969} C_VEL
LIN {X 0,Y 301.168,Z 600.544,A -85,B 0,C 180,E1 -16373.3,E2 -16373.3} C_VEL
LIN {X 0,Y 300.65,Z 600.835,A -85,B 0,C 180,E1 -16374.635,E2 -16374.635} C_VEL
LIN {X 0,Y 300.157,Z 600.733,A -85,B 0,C 180,E1 -16375.972,E2 -16375.972} C_VEL
LIN {X 0,Y 299.612,Z 600.243,A -85,B 0,C 180,E1 -16377.311,E2 -16377.311} C_VEL
LIN {X 0,Y 299.282,Z 599.273,A -85,B 0,C 180,E1 -16378.654,E2 -16378.654} C_VEL
LIN {X 0,Y 298.838,Z 597.89,A -85,B 0,C 180,E1 -16380,E2 -16380} C_VEL
LIN {X 0,Y 298.691,Z 594.946,A -85,B 0,C 180,E1 -16382.023,E2 -16382.023} C_VEL
LIN {X 0,Y 298.548,Z 590.96,A -85,B 0,C 180,E1 -16384.05,E2 -16384.05} C_VEL
LIN {X 0,Y 298.762,Z 585.805,A -85,B 0,C 180,E1 -16386.077,E2 -16386.077} C_VEL
LIN {X 0,Y 299.084,Z 579.332,A -85,B 0,C 180,E1 -16388.105,E2 -16388.105} C_VEL
LIN {X 0,Y 299.535,Z 571.571,A -85,B 0,C 180,E1 -16390.067,E2 -16390.067} C_VEL
LIN {X 0,Y 299.973,Z 563.113,A -85,B 0,C 180,E1 -16391.83,E2 -16391.83} C_VEL
LIN {X 0,Y 300.593,Z 553.304,A -85,B 0,C 180,E1 -16393.521,E2 -16393.521} C_VEL
LIN {X 0,Y 301.171,Z 542.465,A -85,B 0,C 180,E1 -16395.047,E2 -16395.047} C_VEL
LIN {X 0,Y 301.881,Z 530.645,A -85,B 0,C 180,E1 -16396.396,E2 -16396.396} C_VEL
LIN {X 0,Y 302.409,Z 517.409,A -85,B 0,C 180,E1 -16397.585,E2 -16397.585} C_VEL
LIN {X 0,Y 302.848,Z 504.338,A -85,B 0,C 180,E1 -16398.476,E2 -16398.476} C_VEL
LIN {X 0,Y 303.176,Z 490.003,A -85,B 0,C 180,E1 -16399.157,E2 -16399.157} C_VEL
LIN {X 0,Y 304.068,Z 448.956,A -85,B 0,C 180,E1 -16400.568,E2 -16400.568} C_VEL
LIN {X 0,Y 304.522,Z 431.576,A -85,B 0,C 180,E1 -16401.16,E2 -16401.16} C_VEL
LIN {X 0,Y 298.659,Z 412.173,A -85,B 0,C 180,E1 -16402.118,E2 -16402.118} C_VEL
LIN {X 0,Y 298.524,Z 411.369,A -85,B 0,C 180,E1 -16402.377,E2 -16402.377} C_VEL
LIN {X 0,Y 298.414,Z 411.311,A -85,B 0,C 180,E1 -16406.582,E2 -16406.582} C_VEL
LIN {X 0,Y 298.399,Z 411.299,A -85,B 0,C 180,E1 -16409.644,E2 -16409.644} C_VEL
LIN {X 0,Y 298.394,Z 411.304,A -85,B 0,C 180,E1 -16412.801,E2 -16412.801} C_VEL
LIN {X 0,Y 298.446,Z 411.306,A -85,B 0,C 180,E1 -16416.807,E2 -16416.807} C_VEL
LIN {X 0,Y 298.388,Z 411.312,A -85,B 0,C 180,E1 -16421.088,E2 -16421.088} C_VEL
LIN {X 0,Y 298.4,Z 411.311,A -85,B 0,C 180,E1 -16423.103,E2 -16423.103} C_VEL
LIN {X 0,Y 298.423,Z 411.323,A -85,B 0,C 180,E1 -16427.888,E2 -16427.888} C_VEL
LIN {X 0,Y 298.463,Z 411.697,A -85,B 0,C 180,E1 -16428.29,E2 -16428.29} C_VEL
LIN {X 0,Y 302.924,Z 424.856,A -85,B 0,C 180,E1 -16431.541,E2 -16431.541} C_VEL
LIN {X 0,Y 306.499,Z 437.335,A -85,B 0,C 180,E1 -16434.39,E2 -16434.39} C_VEL
LIN {X 0,Y 309.62,Z 450.795,A -85,B 0,C 180,E1 -16437.275,E2 -16437.275} C_VEL
LIN {X 0,Y 310.098,Z 454.091,A -85,B 0,C 180,E1 -16437.934,E2 -16437.934} C_VEL
LIN {X 0,Y 307.947,Z 475.596,A -85,B 0,C 180,E1 -16441.549,E2 -16441.549} C_VEL
LIN {X 0,Y 306.913,Z 487.97,A -85,B 0,C 180,E1 -16443.527,E2 -16443.527} C_VEL
LIN {X 0,Y 311.494,Z 521.082,A -85,B 0,C 180,E1 -16444.794,E2 -16444.794} C_VEL
LIN {X 0,Y 309.545,Z 599.916,A -85,B 0,C 180,E1 -16446.633,E2 -16446.633} C_VEL
LIN {X 0,Y 308.733,Z 612.699,A -85,B 0,C 180,E1 -16447.144,E2 -16447.144} C_VEL
LIN {X 0,Y 307.703,Z 625.543,A -85,B 0,C 180,E1 -16447.949,E2 -16447.949} C_VEL
LIN {X 0,Y 306.292,Z 637.806,A -85,B 0,C 180,E1 -16448.991,E2 -16448.991} C_VEL
LIN {X 0,Y 304.906,Z 648.108,A -85,B 0,C 180,E1 -16450.124,E2 -16450.124} C_VEL
LIN {X 0,Y 303.559,Z 657.552,A -85,B 0,C 180,E1 -16451.423,E2 -16451.423} C_VEL
LIN {X 0,Y 302.066,Z 667.331,A -85,B 0,C 180,E1 -16453.092,E2 -16453.092} C_VEL
LIN {X 0,Y 300.427,Z 676.744,A -85,B 0,C 180,E1 -16455.089,E2 -16455.089} C_VEL
LIN {X 0,Y 299.132,Z 684.219,A -85,B 0,C 180,E1 -16457.103,E2 -16457.103} C_VEL
LIN {X 0,Y 298.135,Z 690.218,A -85,B 0,C 180,E1 -16459.13,E2 -16459.13} C_VEL
LIN {X 0,Y 297.399,Z 694.964,A -85,B 0,C 180,E1 -16461.164,E2 -16461.164} C_VEL
LIN {X 0,Y 296.947,Z 698.595,A -85,B 0,C 180,E1 -16463.204,E2 -16463.204} C_VEL
LIN {X 0,Y 296.707,Z 700.465,A -85,B 0,C 180,E1 -16464.563,E2 -16464.563} C_VEL
LIN {X 0,Y 296.609,Z 701.892,A -85,B 0,C 180,E1 -16465.924,E2 -16465.924} C_VEL
LIN {X 0,Y 296.546,Z 702.892,A -85,B 0,C 180,E1 -16467.283,E2 -16467.283} C_VEL
LIN {X 0,Y 296.453,Z 703.743,A -85,B 0,C 180,E1 -16470,E2 -16470} C_VEL
LIN {X 0,Y 296.461,Z 703.547,A -85,B 0,C 180,E1 -16471.359,E2 -16471.359} C_VEL
LIN {X 0,Y 296.545,Z 702.956,A -85,B 0,C 180,E1 -16472.717,E2 -16472.717} C_VEL
LIN {X 0,Y 296.604,Z 701.981,A -85,B 0,C 180,E1 -16474.077,E2 -16474.077} C_VEL
LIN {X 0,Y 296.756,Z 699.995,A -85,B 0,C 180,E1 -16475.912,E2 -16475.912} C_VEL
LIN {X 0,Y 297.171,Z 696.501,A -85,B 0,C 180,E1 -16478.158,E2 -16478.158} C_VEL
LIN {X 0,Y 297.815,Z 692.204,A -85,B 0,C 180,E1 -16480.195,E2 -16480.195} C_VEL
LIN {X 0,Y 298.741,Z 686.715,A -85,B 0,C 180,E1 -16482.224,E2 -16482.224} C_VEL
LIN {X 0,Y 299.888,Z 679.832,A -85,B 0,C 180,E1 -16484.245,E2 -16484.245} C_VEL
LIN {X 0,Y 301.447,Z 671.224,A -85,B 0,C 180,E1 -16486.247,E2 -16486.247} C_VEL
LIN {X 0,Y 302.958,Z 661.483,A -85,B 0,C 180,E1 -16488.068,E2 -16488.068} C_VEL
LIN {X 0,Y 304.439,Z 651.446,A -85,B 0,C 180,E1 -16489.557,E2 -16489.557} C_VEL
LIN {X 0,Y 306.003,Z 640.419,A -85,B 0,C 180,E1 -16490.854,E2 -16490.854} C_VEL
LIN {X 0,Y 307.245,Z 629.999,A -85,B 0,C 180,E1 -16491.821,E2 -16491.821} C_VEL
LIN {X 0,Y 308.419,Z 617.444,A -85,B 0,C 180,E1 -16492.704,E2 -16492.704} C_VEL
LIN {X 0,Y 309.385,Z 604.106,A -85,B 0,C 180,E1 -16493.336,E2 -16493.336} C_VEL
LIN {X 0,Y 310.014,Z 588.024,A -85,B 0,C 180,E1 -16493.772,E2 -16493.772} C_VEL
LIN {X 0,Y 311.544,Z 520.745,A -85,B 0,C 180,E1 -16495.325,E2 -16495.325} C_VEL
LIN {X 0,Y 307.015,Z 488.473,A -85,B 0,C 180,E1 -16496.557,E2 -16496.557} C_VEL
LIN {X 0,Y 307.039,Z 486.593,A -85,B 0,C 180,E1 -16496.786,E2 -16496.786} C_VEL
LIN {X 0,Y 308.815,Z 467.004,A -85,B 0,C 180,E1 -16500.001,E2 -16500.001} C_VEL
LIN {X 0,Y 308.582,Z 462.87,A -85,B 0,C 180,E1 -16500.78,E2 -16500.78} C_VEL
LIN {X 0,Y 307.32,Z 459.094,A -85,B 0,C 180,E1 -16501.602,E2 -16501.602} C_VEL
LIN {X 0,Y 303.622,Z 451.979,A -85,B 0,C 180,E1 -16503.311,E2 -16503.311} C_VEL
LIN {X 0,Y 301.776,Z 446.959,A -85,B 0,C 180,E1 -16504.472,E2 -16504.472} C_VEL
LIN {X 0,Y 298.521,Z 434.055,A -85,B 0,C 180,E1 -16507.386,E2 -16507.386} C_VEL
LIN {X 0,Y 295.299,Z 423.804,A -85,B 0,C 180,E1 -16509.867,E2 -16509.867} C_VEL
LIN {X 0,Y 291.375,Z 412.409,A -85,B 0,C 180,E1 -16512.806,E2 -16512.806} C_VEL
LIN {X 0,Y 291.291,Z 412.184,A -85,B 0,C 180,E1 -16516.371,E2 -16516.371} C_VEL
LIN {X 0,Y 291.358,Z 412.194,A -85,B 0,C 180,E1 -16520.524,E2 -16520.524} C_VEL
LIN {X 0,Y 291.392,Z 412.177,A -85,B 0,C 180,E1 -16522.917,E2 -16522.917} C_VEL
LIN {X 0,Y 291.346,Z 412.18,A -85,B 0,C 180,E1 -16526.302,E2 -16526.302} C_VEL
LIN {X 0,Y 291.338,Z 412.185,A -85,B 0,C 180,E1 -16530.278,E2 -16530.278} C_VEL
LIN {X 0,Y 291.361,Z 412.192,A -85,B 0,C 180,E1 -16534.266,E2 -16534.266} C_VEL
LIN {X 0,Y 291.366,Z 412.176,A -85,B 0,C 180,E1 -16537.298,E2 -16537.298} C_VEL
LIN {X 0,Y 291.393,Z 412.183,A -85,B 0,C 180,E1 -16540.265,E2 -16540.265} C_VEL
LIN {X 0,Y 291.477,Z 412.176,A -85,B 0,C 180,E1 -16544.683,E2 -16544.683} C_VEL
LIN {X 0,Y 291.529,Z 412.144,A -85,B 0,C 180,E1 -16548.88,E2 -16548.88} C_VEL
LIN {X 0,Y 291.655,Z 412.155,A -85,B 0,C 180,E1 -16551.687,E2 -16551.687} C_VEL
LIN {X 0,Y 291.599,Z 412.139,A -85,B 0,C 180,E1 -16554.468,E2 -16554.468} C_VEL
LIN {X 0,Y 291.874,Z 412.127,A -85,B 0,C 180,E1 -16558.62,E2 -16558.62} C_VEL
LIN {X 0,Y 291.872,Z 412.105,A -85,B 0,C 180,E1 -16561.38,E2 -16561.38} C_VEL
LIN {X 0,Y 291.69,Z 412.149,A -85,B 0,C 180,E1 -16566.919,E2 -16566.919} C_VEL
LIN {X 0,Y 291.57,Z 412.138,A -85,B 0,C 180,E1 -16569.714,E2 -16569.714} C_VEL
LIN {X 0,Y 291.479,Z 412.173,A -85,B 0,C 180,E1 -16573.952,E2 -16573.952} C_VEL
LIN {X 0,Y 291.382,Z 412.162,A -85,B 0,C 180,E1 -16576.824,E2 -16576.824} C_VEL
LIN {X 0,Y 291.394,Z 412.19,A -85,B 0,C 180,E1 -16579.842,E2 -16579.842} C_VEL
LIN {X 0,Y 291.328,Z 412.178,A -85,B 0,C 180,E1 -16584.212,E2 -16584.212} C_VEL
LIN {X 0,Y 291.331,Z 412.189,A -85,B 0,C 180,E1 -16587.281,E2 -16587.281} C_VEL
LIN {X 0,Y 291.304,Z 412.188,A -85,B 0,C 180,E1 -16590.441,E2 -16590.441} C_VEL
LIN {X 0,Y 291.346,Z 412.179,A -85,B 0,C 180,E1 -16593.698,E2 -16593.698} C_VEL
LIN {X 0,Y 291.355,Z 412.194,A -85,B 0,C 180,E1 -16597.248,E2 -16597.248} C_VEL
LIN {X 0,Y 291.301,Z 412.142,A -85,B 0,C 180,E1 -16600.648,E2 -16600.648} C_VEL
LIN {X 0,Y 291.283,Z 412.19,A -85,B 0,C 180,E1 -16604.403,E2 -16604.403} C_VEL
LIN {X 0,Y 291.295,Z 412.156,A -85,B 0,C 180,E1 -16608.411,E2 -16608.411} C_VEL
LIN {X 0,Y 291.438,Z 412.346,A -85,B 0,C 180,E1 -16612.895,E2 -16612.895} C_VEL
LIN {X 0,Y 294.703,Z 427.792,A -85,B 0,C 180,E1 -16616.736,E2 -16616.736} C_VEL
LIN {X 0,Y 295.848,Z 433.282,A -85,B 0,C 180,E1 -16617.97,E2 -16617.97} C_VEL
LIN {X 0,Y 298.47,Z 441.987,A -85,B 0,C 180,E1 -16619.024,E2 -16619.024} C_VEL
LIN {X 0,Y 299.574,Z 461.657,A -85,B 0,C 180,E1 -16620.702,E2 -16620.702} C_VEL
LIN {X 0,Y 300.34,Z 487.807,A -85,B 0,C 180,E1 -16622.935,E2 -16622.935} C_VEL
LIN {X 0,Y 303.447,Z 516.409,A -85,B 0,C 180,E1 -16624.012,E2 -16624.012} C_VEL
LIN {X 0,Y 304.455,Z 529.611,A -85,B 0,C 180,E1 -16624.443,E2 -16624.443} C_VEL
LIN {X 0,Y 302.574,Z 604.158,A -85,B 0,C 180,E1 -16626.198,E2 -16626.198} C_VEL
LIN {X 0,Y 301.756,Z 616.536,A -85,B 0,C 180,E1 -16626.675,E2 -16626.675} C_VEL
LIN {X 0,Y 300.716,Z 628.67,A -85,B 0,C 180,E1 -16627.408,E2 -16627.408} C_VEL
LIN {X 0,Y 299.389,Z 641.4,A -85,B 0,C 180,E1 -16628.482,E2 -16628.482} C_VEL
LIN {X 0,Y 297.902,Z 651.981,A -85,B 0,C 180,E1 -16629.636,E2 -16629.636} C_VEL
LIN {X 0,Y 296.212,Z 662.765,A -85,B 0,C 180,E1 -16631.139,E2 -16631.139} C_VEL
LIN {X 0,Y 294.632,Z 672.806,A -85,B 0,C 180,E1 -16632.907,E2 -16632.907} C_VEL
LIN {X 0,Y 293.255,Z 681.058,A -85,B 0,C 180,E1 -16634.715,E2 -16634.715} C_VEL
LIN {X 0,Y 291.855,Z 688.602,A -85,B 0,C 180,E1 -16636.775,E2 -16636.775} C_VEL
LIN {X 0,Y 290.886,Z 694.658,A -85,B 0,C 180,E1 -16638.855,E2 -16638.855} C_VEL
LIN {X 0,Y 290.192,Z 699.439,A -85,B 0,C 180,E1 -16640.943,E2 -16640.943} C_VEL
LIN {X 0,Y 289.761,Z 703.087,A -85,B 0,C 180,E1 -16643.034,E2 -16643.034} C_VEL
LIN {X 0,Y 289.605,Z 704.967,A -85,B 0,C 180,E1 -16644.429,E2 -16644.429} C_VEL
LIN {X 0,Y 289.505,Z 706.383,A -85,B 0,C 180,E1 -16645.823,E2 -16645.823} C_VEL
LIN {X 0,Y 289.488,Z 707.383,A -85,B 0,C 180,E1 -16647.217,E2 -16647.217} C_VEL
LIN {X 0,Y 289.438,Z 707.993,A -85,B 0,C 180,E1 -16648.608,E2 -16648.608} C_VEL
LIN {X 0,Y 289.447,Z 708.209,A -85,B 0,C 180,E1 -16650,E2 -16650} C_VEL
LIN {X 0,Y 289.463,Z 707.986,A -85,B 0,C 180,E1 -16651.391,E2 -16651.391} C_VEL
LIN {X 0,Y 289.518,Z 707.371,A -85,B 0,C 180,E1 -16652.783,E2 -16652.783} C_VEL
LIN {X 0,Y 289.54,Z 706.366,A -85,B 0,C 180,E1 -16654.176,E2 -16654.176} C_VEL
LIN {X 0,Y 289.63,Z 704.649,A -85,B 0,C 180,E1 -16655.798,E2 -16655.798} C_VEL
LIN {X 0,Y 290.013,Z 700.739,A -85,B 0,C 180,E1 -16658.36,E2 -16658.36} C_VEL
LIN {X 0,Y 290.633,Z 696.343,A -85,B 0,C 180,E1 -16660.449,E2 -16660.449} C_VEL
LIN {X 0,Y 291.49,Z 690.734,A -85,B 0,C 180,E1 -16662.532,E2 -16662.532} C_VEL
LIN {X 0,Y 292.777,Z 683.67,A -85,B 0,C 180,E1 -16664.599,E2 -16664.599} C_VEL
LIN {X 0,Y 294.234,Z 674.843,A -85,B 0,C 180,E1 -16666.656,E2 -16666.656} C_VEL
LIN {X 0,Y 295.887,Z 664.729,A -85,B 0,C 180,E1 -16668.523,E2 -16668.523} C_VEL
LIN {X 0,Y 297.504,Z 654.386,A -85,B 0,C 180,E1 -16670.031,E2 -16670.031} C_VEL
LIN {X 0,Y 299.094,Z 642.871,A -85,B 0,C 180,E1 -16671.359,E2 -16671.359} C_VEL
LIN {X 0,Y 300.523,Z 630.574,A -85,B 0,C 180,E1 -16672.425,E2 -16672.425} C_VEL
LIN {X 0,Y 301.347,Z 622.82,A -85,B 0,C 180,E1 -16672.994,E2 -16672.994} C_VEL
LIN {X 0,Y 304.758,Z 610.541,A -85,B 0,C 180,E1 -16674.525,E2 -16674.525} C_VEL
LIN {X 0,Y 308.172,Z 596.83,A -85,B 0,C 180,E1 -16675.859,E2 -16675.859} C_VEL
LIN {X 0,Y 311.118,Z 582.404,A -85,B 0,C 180,E1 -16676.949,E2 -16676.949} C_VEL
LIN {X 0,Y 313.559,Z 567.983,A -85,B 0,C 180,E1 -16677.761,E2 -16677.761} C_VEL
LIN {X 0,Y 316.666,Z 539.179,A -85,B 0,C 180,E1 -16678.938,E2 -16678.938} C_VEL
LIN {X 0,Y 317.459,Z 530.421,A -85,B 0,C 180,E1 -16679.308,E2 -16679.308} C_VEL
LIN {X 0,Y 317.849,Z 514.993,A -85,B 0,C 180,E1 -16680.199,E2 -16680.199} C_VEL
LIN {X 0,Y 317.532,Z 501.08,A -85,B 0,C 180,E1 -16681.208,E2 -16681.208} C_VEL
LIN {X 0,Y 316.663,Z 486.847,A -85,B 0,C 180,E1 -16682.461,E2 -16682.461} C_VEL
LIN {X 0,Y 315.434,Z 473.23,A -85,B 0,C 180,E1 -16683.908,E2 -16683.908} C_VEL
LIN {X 0,Y 314.64,Z 466.17,A -85,B 0,C 180,E1 -16684.778,E2 -16684.778} C_VEL
LIN {X 0,Y 313.202,Z 461.92,A -85,B 0,C 180,E1 -16685.691,E2 -16685.691} C_VEL
LIN {X 0,Y 309.885,Z 453.359,A -85,B 0,C 180,E1 -16688.047,E2 -16688.047} C_VEL
LIN {X 0,Y 306.861,Z 446.199,A -85,B 0,C 180,E1 -16691.017,E2 -16691.017} C_VEL
LIN {X 0,Y 305.517,Z 442.275,A -85,B 0,C 180,E1 -16693.357,E2 -16693.357} C_VEL
LIN {X 0,Y 305.065,Z 439.987,A -85,B 0,C 180,E1 -16695.428,E2 -16695.428} C_VEL
LIN {X 0,Y 305.526,Z 438.37,A -85,B 0,C 180,E1 -16697.889,E2 -16697.889} C_VEL
LIN {X 0,Y 306.202,Z 437.975,A -85,B 0,C 180,E1 -16699.237,E2 -16699.237} C_VEL
LIN {X 0,Y 307.897,Z 438.542,A -85,B 0,C 180,E1 -16701.36,E2 -16701.36} C_VEL
LIN {X 0,Y 310.091,Z 439.49,A -85,B 0,C 180,E1 -16703.166,E2 -16703.166} C_VEL
LIN {X 0,Y 313.293,Z 442.194,A -85,B 0,C 180,E1 -16705.241,E2 -16705.241} C_VEL
LIN {X 0,Y 315.954,Z 444.963,A -85,B 0,C 180,E1 -16706.69,E2 -16706.69} C_VEL
LIN {X 0,Y 318.371,Z 448.004,A -85,B 0,C 180,E1 -16707.889,E2 -16707.889} C_VEL
LIN {X 0,Y 322.798,Z 456.223,A -85,B 0,C 180,E1 -16709.914,E2 -16709.914} C_VEL
LIN {X 0,Y 323.996,Z 458.78,A -85,B 0,C 180,E1 -16710.418,E2 -16710.418} C_VEL
LIN {X 0,Y 320.03,Z 492.164,A -85,B 0,C 180,E1 -16711.814,E2 -16711.814} C_VEL
LIN {X 0,Y 318.39,Z 512.148,A -85,B 0,C 180,E1 -16712.783,E2 -16712.783} C_VEL
LIN {X 0,Y 316.961,Z 525.439,A -85,B 0,C 180,E1 -16713.675,E2 -16713.675} C_VEL
LIN {X 0,Y 315.151,Z 537.733,A -85,B 0,C 180,E1 -16714.755,E2 -16714.755} C_VEL
LIN {X 0,Y 313.139,Z 548.936,A -85,B 0,C 180,E1 -16715.996,E2 -16715.996} C_VEL
LIN {X 0,Y 310.778,Z 559.135,A -85,B 0,C 180,E1 -16717.391,E2 -16717.391} C_VEL
LIN {X 0,Y 308.315,Z 568.75,A -85,B 0,C 180,E1 -16719.039,E2 -16719.039} C_VEL
LIN {X 0,Y 306.187,Z 576.039,A -85,B 0,C 180,E1 -16720.559,E2 -16720.559} C_VEL
LIN {X 0,Y 303.679,Z 583.5,A -85,B 0,C 180,E1 -16722.491,E2 -16722.491} C_VEL
LIN {X 0,Y 301.362,Z 589.485,A -85,B 0,C 180,E1 -16724.443,E2 -16724.443} C_VEL
LIN {X 0,Y 299.282,Z 594.201,A -85,B 0,C 180,E1 -16726.418,E2 -16726.418} C_VEL
LIN {X 0,Y 298.081,Z 596.687,A -85,B 0,C 180,E1 -16727.749,E2 -16727.749} C_VEL
LIN {X 0,Y 296.961,Z 598.646,A -85,B 0,C 180,E1 -16729.086,E2 -16729.086} C_VEL
LIN {X 0,Y 295.929,Z 600.177,A -85,B 0,C 180,E1 -16730.431,E2 -16730.431} C_VEL
LIN {X 0,Y 294.979,Z 601.302,A -85,B 0,C 180,E1 -16731.781,E2 -16731.781} C_VEL
LIN {X 0,Y 294.258,Z 601.919,A -85,B 0,C 180,E1 -16733.141,E2 -16733.141} C_VEL
LIN {X 0,Y 293.699,Z 602.11,A -85,B 0,C 180,E1 -16734.507,E2 -16734.507} C_VEL
LIN {X 0,Y 293.186,Z 601.901,A -85,B 0,C 180,E1 -16735.876,E2 -16735.876} C_VEL
LIN {X 0,Y 292.605,Z 601.261,A -85,B 0,C 180,E1 -16737.247,E2 -16737.247} C_VEL
LIN {X 0,Y 292.248,Z 600.169,A -85,B 0,C 180,E1 -16738.622,E2 -16738.622} C_VEL
LIN {X 0,Y 291.809,Z 598.685,A -85,B 0,C 180,E1 -16740,E2 -16740} C_VEL
LIN {X 0,Y 291.631,Z 595.557,A -85,B 0,C 180,E1 -16742.072,E2 -16742.072} C_VEL
LIN {X 0,Y 291.487,Z 591.37,A -85,B 0,C 180,E1 -16744.148,E2 -16744.148} C_VEL
LIN {X 0,Y 291.767,Z 584.943,A -85,B 0,C 180,E1 -16746.57,E2 -16746.57} C_VEL
LIN {X 0,Y 292.123,Z 578.128,A -85,B 0,C 180,E1 -16748.61,E2 -16748.61} C_VEL
LIN {X 0,Y 292.6,Z 569.398,A -85,B 0,C 180,E1 -16750.728,E2 -16750.728} C_VEL
LIN {X 0,Y 293.21,Z 558.682,A -85,B 0,C 180,E1 -16752.81,E2 -16752.81} C_VEL
LIN {X 0,Y 293.843,Z 547.534,A -85,B 0,C 180,E1 -16754.545,E2 -16754.545} C_VEL
LIN {X 0,Y 294.483,Z 536.629,A -85,B 0,C 180,E1 -16755.93,E2 -16755.93} C_VEL
LIN {X 0,Y 295.143,Z 525.291,A -85,B 0,C 180,E1 -16757.098,E2 -16757.098} C_VEL
LIN {X 0,Y 295.617,Z 511.806,A -85,B 0,C 180,E1 -16758.182,E2 -16758.182} C_VEL
LIN {X 0,Y 295.928,Z 498.607,A -85,B 0,C 180,E1 -16758.97,E2 -16758.97} C_VEL
LIN {X 0,Y 296.296,Z 478.362,A -85,B 0,C 180,E1 -16759.755,E2 -16759.755} C_VEL
LIN {X 0,Y 297.542,Z 432.95,A -85,B 0,C 180,E1 -16761.364,E2 -16761.364} C_VEL
LIN {X 0,Y 291.664,Z 413.191,A -85,B 0,C 180,E1 -16762.353,E2 -16762.353} C_VEL
LIN {X 0,Y 291.47,Z 412.27,A -85,B 0,C 180,E1 -16762.614,E2 -16762.614} C_VEL
LIN {X 0,Y 291.36,Z 412.183,A -85,B 0,C 180,E1 -16767.278,E2 -16767.278} C_VEL
LIN {X 0,Y 291.322,Z 412.19,A -85,B 0,C 180,E1 -16770.439,E2 -16770.439} C_VEL
LIN {X 0,Y 291.345,Z 412.176,A -85,B 0,C 180,E1 -16773.699,E2 -16773.699} C_VEL
LIN {X 0,Y 291.374,Z 412.182,A -85,B 0,C 180,E1 -16777.253,E2 -16777.253} C_VEL
LIN {X 0,Y 291.334,Z 412.195,A -85,B 0,C 180,E1 -16780.643,E2 -16780.643} C_VEL
LIN {X 0,Y 291.292,Z 412.196,A -85,B 0,C 180,E1 -16784.402,E2 -16784.402} C_VEL
LIN {X 0,Y 291.397,Z 412.375,A -85,B 0,C 180,E1 -16787.32,E2 -16787.32} C_VEL
LIN {X 0,Y 296.269,Z 426.637,A -85,B 0,C 180,E1 -16790.976,E2 -16790.976} C_VEL
LIN {X 0,Y 300.116,Z 440.211,A -85,B 0,C 180,E1 -16794.166,E2 -16794.166} C_VEL
LIN {X 0,Y 302.991,Z 452.656,A -85,B 0,C 180,E1 -16796.869,E2 -16796.869} C_VEL
LIN {X 0,Y 303.536,Z 456.092,A -85,B 0,C 180,E1 -16797.575,E2 -16797.575} C_VEL
LIN {X 0,Y 301.399,Z 476.591,A -85,B 0,C 180,E1 -16801.063,E2 -16801.063} C_VEL
LIN {X 0,Y 300.426,Z 488.278,A -85,B 0,C 180,E1 -16802.928,E2 -16802.928} C_VEL
LIN {X 0,Y 305.033,Z 521.245,A -85,B 0,C 180,E1 -16804.226,E2 -16804.226} C_VEL
LIN {X 0,Y 303.177,Z 597.277,A -85,B 0,C 180,E1 -16806.021,E2 -16806.021} C_VEL
LIN {X 0,Y 302.33,Z 611.035,A -85,B 0,C 180,E1 -16806.541,E2 -16806.541} C_VEL
LIN {X 0,Y 301.301,Z 623.388,A -85,B 0,C 180,E1 -16807.274,E2 -16807.274} C_VEL
LIN {X 0,Y 300.122,Z 634.451,A -85,B 0,C 180,E1 -16808.177,E2 -16808.177} C_VEL
LIN {X 0,Y 298.643,Z 645.4,A -85,B 0,C 180,E1 -16809.329,E2 -16809.329} C_VEL
LIN {X 0,Y 296.929,Z 656.696,A -85,B 0,C 180,E1 -16810.846,E2 -16810.846} C_VEL
LIN {X 0,Y 295.536,Z 665.629,A -85,B 0,C 180,E1 -16812.35,E2 -16812.35} C_VEL
LIN {X 0,Y 294.127,Z 673.89,A -85,B 0,C 180,E1 -16814.051,E2 -16814.051} C_VEL
LIN {X 0,Y 292.575,Z 681.947,A -85,B 0,C 180,E1 -16816.101,E2 -16816.101} C_VEL
LIN {X 0,Y 291.48,Z 688.429,A -85,B 0,C 180,E1 -16818.174,E2 -16818.174} C_VEL
LIN {X 0,Y 290.586,Z 693.584,A -85,B 0,C 180,E1 -16820.253,E2 -16820.253} C_VEL
LIN {X 0,Y 290.032,Z 697.576,A -85,B 0,C 180,E1 -16822.341,E2 -16822.341} C_VEL
LIN {X 0,Y 289.645,Z 700.52,A -85,B 0,C 180,E1 -16824.43,E2 -16824.43} C_VEL
LIN {X 0,Y 289.514,Z 701.946,A -85,B 0,C 180,E1 -16825.824,E2 -16825.824} C_VEL
LIN {X 0,Y 289.454,Z 702.946,A -85,B 0,C 180,E1 -16827.217,E2 -16827.217} C_VEL
LIN {X 0,Y 289.373,Z 703.797,A -85,B 0,C 180,E1 -16830,E2 -16830} C_VEL
LIN {X 0,Y 289.385,Z 703.601,A -85,B 0,C 180,E1 -16831.392,E2 -16831.392} C_VEL
LIN {X 0,Y 289.453,Z 703.009,A -85,B 0,C 180,E1 -16832.784,E2 -16832.784} C_VEL
LIN {X 0,Y 289.508,Z 702.034,A -85,B 0,C 180,E1 -16834.177,E2 -16834.177} C_VEL
LIN {X 0,Y 289.675,Z 700.266,A -85,B 0,C 180,E1 -16835.883,E2 -16835.883} C_VEL
LIN {X 0,Y 290.128,Z 696.554,A -85,B 0,C 180,E1 -16838.357,E2 -16838.357} C_VEL
LIN {X 0,Y 290.81,Z 692.256,A -85,B 0,C 180,E1 -16840.443,E2 -16840.443} C_VEL
LIN {X 0,Y 291.786,Z 686.765,A -85,B 0,C 180,E1 -16842.52,E2 -16842.52} C_VEL
LIN {X 0,Y 293.011,Z 679.88,A -85,B 0,C 180,E1 -16844.587,E2 -16844.587} C_VEL
LIN {X 0,Y 294.626,Z 671.271,A -85,B 0,C 180,E1 -16846.634,E2 -16846.634} C_VEL
LIN {X 0,Y 296.051,Z 662.453,A -85,B 0,C 180,E1 -16848.333,E2 -16848.333} C_VEL
LIN {X 0,Y 297.542,Z 652.734,A -85,B 0,C 180,E1 -16849.849,E2 -16849.849} C_VEL
LIN {X 0,Y 299.183,Z 641.978,A -85,B 0,C 180,E1 -16851.172,E2 -16851.172} C_VEL
LIN {X 0,Y 300.653,Z 630.025,A -85,B 0,C 180,E1 -16852.325,E2 -16852.325} C_VEL
LIN {X 0,Y 301.753,Z 618.819,A -85,B 0,C 180,E1 -16853.143,E2 -16853.143} C_VEL
LIN {X 0,Y 302.749,Z 606.144,A -85,B 0,C 180,E1 -16853.788,E2 -16853.788} C_VEL
LIN {X 0,Y 303.421,Z 591.506,A -85,B 0,C 180,E1 -16854.231,E2 -16854.231} C_VEL
LIN {X 0,Y 305.145,Z 521.791,A -85,B 0,C 180,E1 -16855.866,E2 -16855.866} C_VEL
LIN {X 0,Y 300.617,Z 489.264,A -85,B 0,C 180,E1 -16857.139,E2 -16857.139} C_VEL
LIN {X 0,Y 300.449,Z 487.488,A -85,B 0,C 180,E1 -16857.266,E2 -16857.266} C_VEL
LIN {X 0,Y 302.943,Z 462.405,A -85,B 0,C 180,E1 -16861.465,E2 -16861.465} C_VEL
LIN {X 0,Y 303.53,Z 455.318,A -85,B 0,C 180,E1 -16862.708,E2 -16862.708} C_VEL
LIN {X 0,Y 301.776,Z 446.959,A -85,B 0,C 180,E1 -16864.472,E2 -16864.472} C_VEL
LIN {X 0,Y 300.331,Z 443.451,A -85,B 0,C 180,E1 -16865.331,E2 -16865.331} C_VEL
LIN {X 0,Y 296.279,Z 438.656,A -85,B 0,C 180,E1 -16866.805,E2 -16866.805} C_VEL
LIN {X 0,Y 292.799,Z 434.966,A -85,B 0,C 180,E1 -16868.015,E2 -16868.015} C_VEL
LIN {X 0,Y 290.776,Z 431.805,A -85,B 0,C 180,E1 -16868.928,E2 -16868.928} C_VEL
LIN {X 0,Y 290.309,Z 430.605,A -85,B 0,C 180,E1 -16869.229,E2 -16869.229} C_VEL
LIN {X 0,Y 285.442,Z 416.499,A -85,B 0,C 180,E1 -16872.838,E2 -16872.838} C_VEL
LIN {X 0,Y 284.289,Z 413.217,A -85,B 0,C 180,E1 -16873.805,E2 -16873.805} C_VEL
LIN {X 0,Y 284.242,Z 413.08,A -85,B 0,C 180,E1 -16878.119,E2 -16878.119} C_VEL
LIN {X 0,Y 284.311,Z 413.06,A -85,B 0,C 180,E1 -16882.282,E2 -16882.282} C_VEL
LIN {X 0,Y 284.309,Z 413.065,A -85,B 0,C 180,E1 -16885.351,E2 -16885.351} C_VEL
LIN {X 0,Y 284.281,Z 413.075,A -85,B 0,C 180,E1 -16888.724,E2 -16888.724} C_VEL
LIN {X 0,Y 284.328,Z 413.067,A -85,B 0,C 180,E1 -16892.855,E2 -16892.855} C_VEL
LIN {X 0,Y 284.33,Z 413.048,A -85,B 0,C 180,E1 -16896.704,E2 -16896.704} C_VEL
LIN {X 0,Y 284.326,Z 413.05,A -85,B 0,C 180,E1 -16901.256,E2 -16901.256} C_VEL
LIN {X 0,Y 284.437,Z 413.055,A -85,B 0,C 180,E1 -16905.695,E2 -16905.695} C_VEL
LIN {X 0,Y 284.516,Z 413.027,A -85,B 0,C 180,E1 -16910.043,E2 -16910.043} C_VEL
LIN {X 0,Y 284.645,Z 413.026,A -85,B 0,C 180,E1 -16912.909,E2 -16912.909} C_VEL
LIN {X 0,Y 284.841,Z 413.003,A -85,B 0,C 180,E1 -16918.586,E2 -16918.586} C_VEL
LIN {X 0,Y 284.839,Z 412.98,A -85,B 0,C 180,E1 -16921.414,E2 -16921.414} C_VEL
LIN {X 0,Y 284.645,Z 413.026,A -85,B 0,C 180,E1 -16927.091,E2 -16927.091} C_VEL
LIN {X 0,Y 284.516,Z 413.016,A -85,B 0,C 180,E1 -16929.957,E2 -16929.957} C_VEL
LIN {X 0,Y 284.411,Z 413.051,A -85,B 0,C 180,E1 -16934.306,E2 -16934.306} C_VEL
LIN {X 0,Y 284.331,Z 413.042,A -85,B 0,C 180,E1 -16937.254,E2 -16937.254} C_VEL
LIN {X 0,Y 284.324,Z 413.068,A -85,B 0,C 180,E1 -16940.246,E2 -16940.246} C_VEL
LIN {X 0,Y 284.295,Z 413.05,A -85,B 0,C 180,E1 -16943.84,E2 -16943.84} C_VEL
LIN {X 0,Y 284.288,Z 413.069,A -85,B 0,C 180,E1 -16947.13,E2 -16947.13} C_VEL
LIN {X 0,Y 284.276,Z 413.058,A -85,B 0,C 180,E1 -16950.084,E2 -16950.084} C_VEL
LIN {X 0,Y 284.307,Z 413.064,A -85,B 0,C 180,E1 -16952.945,E2 -16952.945} C_VEL
LIN {X 0,Y 284.32,Z 413.068,A -85,B 0,C 180,E1 -16956.388,E2 -16956.388} C_VEL
LIN {X 0,Y 284.283,Z 413.022,A -85,B 0,C 180,E1 -16959.999,E2 -16959.999} C_VEL
LIN {X 0,Y 284.235,Z 413.06,A -85,B 0,C 180,E1 -16964.187,E2 -16964.187} C_VEL
LIN {X 0,Y 284.24,Z 413.036,A -85,B 0,C 180,E1 -16968.118,E2 -16968.118} C_VEL
LIN {X 0,Y 284.341,Z 413.158,A -85,B 0,C 180,E1 -16972.609,E2 -16972.609} C_VEL
LIN {X 0,Y 287.31,Z 427.018,A -85,B 0,C 180,E1 -16976.167,E2 -16976.167} C_VEL
LIN {X 0,Y 288.206,Z 430.734,A -85,B 0,C 180,E1 -16976.714,E2 -16976.714} C_VEL
LIN {X 0,Y 292.16,Z 443.298,A -85,B 0,C 180,E1 -16978.315,E2 -16978.315} C_VEL
LIN {X 0,Y 292.759,Z 447.951,A -85,B 0,C 180,E1 -16978.772,E2 -16978.772} C_VEL
LIN {X 0,Y 293.808,Z 478.052,A -85,B 0,C 180,E1 -16981.418,E2 -16981.418} C_VEL
LIN {X 0,Y 293.963,Z 488.695,A -85,B 0,C 180,E1 -16982.359,E2 -16982.359} C_VEL
LIN {X 0,Y 297.519,Z 521.769,A -85,B 0,C 180,E1 -16983.593,E2 -16983.593} C_VEL
LIN {X 0,Y 298.064,Z 530.927,A -85,B 0,C 180,E1 -16983.886,E2 -16983.886} C_VEL
LIN {X 0,Y 296.102,Z 604.206,A -85,B 0,C 180,E1 -16985.644,E2 -16985.644} C_VEL
LIN {X 0,Y 295.265,Z 616.537,A -85,B 0,C 180,E1 -16986.131,E2 -16986.131} C_VEL
LIN {X 0,Y 294.182,Z 628.649,A -85,B 0,C 180,E1 -16986.878,E2 -16986.878} C_VEL
LIN {X 0,Y 292.798,Z 641.37,A -85,B 0,C 180,E1 -16987.973,E2 -16987.973} C_VEL
LIN {X 0,Y 291.243,Z 651.944,A -85,B 0,C 180,E1 -16989.149,E2 -16989.149} C_VEL
LIN {X 0,Y 289.478,Z 662.722,A -85,B 0,C 180,E1 -16990.683,E2 -16990.683} C_VEL
LIN {X 0,Y 288.023,Z 671.751,A -85,B 0,C 180,E1 -16992.293,E2 -16992.293} C_VEL
LIN {X 0,Y 286.385,Z 681.01,A -85,B 0,C 180,E1 -16994.339,E2 -16994.339} C_VEL
LIN {X 0,Y 284.903,Z 688.552,A -85,B 0,C 180,E1 -16996.447,E2 -16996.447} C_VEL
LIN {X 0,Y 283.906,Z 694.607,A -85,B 0,C 180,E1 -16998.578,E2 -16998.578} C_VEL
LIN {X 0,Y 283.154,Z 699.387,A -85,B 0,C 180,E1 -17000.715,E2 -17000.715} C_VEL
LIN {X 0,Y 282.691,Z 703.034,A -85,B 0,C 180,E1 -17002.859,E2 -17002.859} C_VEL
LIN {X 0,Y 282.523,Z 704.913,A -85,B 0,C 180,E1 -17004.289,E2 -17004.289} C_VEL
LIN {X 0,Y 282.413,Z 706.329,A -85,B 0,C 180,E1 -17005.718,E2 -17005.718} C_VEL
LIN {X 0,Y 282.395,Z 707.329,A -85,B 0,C 180,E1 -17007.147,E2 -17007.147} C_VEL
LIN {X 0,Y 282.361,Z 707.939,A -85,B 0,C 180,E1 -17008.574,E2 -17008.574} C_VEL
LIN {X 0,Y 282.367,Z 708.155,A -85,B 0,C 180,E1 -17010,E2 -17010} C_VEL
LIN {X 0,Y 282.385,Z 707.932,A -85,B 0,C 180,E1 -17011.426,E2 -17011.426} C_VEL
LIN {X 0,Y 282.424,Z 707.317,A -85,B 0,C 180,E1 -17012.853,E2 -17012.853} C_VEL
LIN {X 0,Y 282.444,Z 706.312,A -85,B 0,C 180,E1 -17014.281,E2 -17014.281} C_VEL
LIN {X 0,Y 282.523,Z 704.885,A -85,B 0,C 180,E1 -17015.71,E2 -17015.71} C_VEL
LIN {X 0,Y 282.814,Z 701.92,A -85,B 0,C 180,E1 -17017.855,E2 -17017.855} C_VEL
LIN {X 0,Y 283.381,Z 697.894,A -85,B 0,C 180,E1 -17019.997,E2 -17019.997} C_VEL
LIN {X 0,Y 284.379,Z 691.684,A -85,B 0,C 180,E1 -17022.488,E2 -17022.488} C_VEL
LIN {X 0,Y 285.661,Z 684.908,A -85,B 0,C 180,E1 -17024.606,E2 -17024.606} C_VEL
LIN {X 0,Y 286.91,Z 677.97,A -85,B 0,C 180,E1 -17026.361,E2 -17026.361} C_VEL
LIN {X 0,Y 288.48,Z 668.774,A -85,B 0,C 180,E1 -17028.252,E2 -17028.252} C_VEL
LIN {X 0,Y 290.044,Z 659.206,A -85,B 0,C 180,E1 -17029.83,E2 -17029.83} C_VEL
LIN {X 0,Y 291.628,Z 648.925,A -85,B 0,C 180,E1 -17031.192,E2 -17031.192} C_VEL
LIN {X 0,Y 293.18,Z 637.614,A -85,B 0,C 180,E1 -17032.368,E2 -17032.368} C_VEL
LIN {X 0,Y 294.591,Z 625.19,A -85,B 0,C 180,E1 -17033.367,E2 -17033.367} C_VEL
LIN {X 0,Y 298.071,Z 613.823,A -85,B 0,C 180,E1 -17034.927,E2 -17034.927} C_VEL
LIN {X 0,Y 301.5,Z 601.36,A -85,B 0,C 180,E1 -17036.289,E2 -17036.289} C_VEL
LIN {X 0,Y 304.797,Z 587.695,A -85,B 0,C 180,E1 -17037.462,E2 -17037.462} C_VEL
LIN {X 0,Y 307.428,Z 574.757,A -85,B 0,C 180,E1 -17038.318,E2 -17038.318} C_VEL
LIN {X 0,Y 309.781,Z 559.267,A -85,B 0,C 180,E1 -17039.101,E2 -17039.101} C_VEL
LIN {X 0,Y 312.75,Z 531.824,A -85,B 0,C 180,E1 -17040.235,E2 -17040.235} C_VEL
LIN {X 0,Y 313.322,Z 516.251,A -85,B 0,C 180,E1 -17041.166,E2 -17041.166} C_VEL
LIN {X 0,Y 313.146,Z 502.599,A -85,B 0,C 180,E1 -17042.209,E2 -17042.209} C_VEL
LIN {X 0,Y 312.538,Z 488.468,A -85,B 0,C 180,E1 -17043.508,E2 -17043.508} C_VEL
LIN {X 0,Y 311.453,Z 473.203,A -85,B 0,C 180,E1 -17045.229,E2 -17045.229} C_VEL
LIN {X 0,Y 311.034,Z 470.136,A -85,B 0,C 180,E1 -17045.683,E2 -17045.683} C_VEL
LIN {X 0,Y 309.835,Z 466.622,A -85,B 0,C 180,E1 -17046.517,E2 -17046.517} C_VEL
LIN {X 0,Y 307.42,Z 459.608,A -85,B 0,C 180,E1 -17048.476,E2 -17048.476} C_VEL
LIN {X 0,Y 304.817,Z 452.945,A -85,B 0,C 180,E1 -17051.268,E2 -17051.268} C_VEL
LIN {X 0,Y 303.637,Z 449.012,A -85,B 0,C 180,E1 -17053.588,E2 -17053.588} C_VEL
LIN {X 0,Y 303.297,Z 446.732,A -85,B 0,C 180,E1 -17055.698,E2 -17055.698} C_VEL
LIN {X 0,Y 303.965,Z 445.089,A -85,B 0,C 180,E1 -17058.343,E2 -17058.343} C_VEL
LIN {X 0,Y 304.836,Z 444.904,A -85,B 0,C 180,E1 -17059.794,E2 -17059.794} C_VEL
LIN {X 0,Y 307.878,Z 446.042,A -85,B 0,C 180,E1 -17062.818,E2 -17062.818} C_VEL
LIN {X 0,Y 311.033,Z 448.821,A -85,B 0,C 180,E1 -17064.999,E2 -17064.999} C_VEL
LIN {X 0,Y 314.024,Z 452.017,A -85,B 0,C 180,E1 -17066.68,E2 -17066.68} C_VEL
LIN {X 0,Y 315.791,Z 454.668,A -85,B 0,C 180,E1 -17067.607,E2 -17067.607} C_VEL
LIN {X 0,Y 319.501,Z 461.97,A -85,B 0,C 180,E1 -17069.441,E2 -17069.441} C_VEL
LIN {X 0,Y 319.302,Z 464.429,A -85,B 0,C 180,E1 -17069.586,E2 -17069.586} C_VEL
LIN {X 0,Y 315.581,Z 494.582,A -85,B 0,C 180,E1 -17070.881,E2 -17070.881} C_VEL
LIN {X 0,Y 313.813,Z 513.144,A -85,B 0,C 180,E1 -17071.817,E2 -17071.817} C_VEL
LIN {X 0,Y 312.033,Z 528.328,A -85,B 0,C 180,E1 -17072.864,E2 -17072.864} C_VEL
LIN {X 0,Y 310.37,Z 538.667,A -85,B 0,C 180,E1 -17073.797,E2 -17073.797} C_VEL
LIN {X 0,Y 307.887,Z 551.011,A -85,B 0,C 180,E1 -17075.201,E2 -17075.201} C_VEL
LIN {X 0,Y 305.388,Z 561.045,A -85,B 0,C 180,E1 -17076.61,E2 -17076.61} C_VEL
LIN {X 0,Y 302.86,Z 570.15,A -85,B 0,C 180,E1 -17078.205,E2 -17078.205} C_VEL
LIN {X 0,Y 300.403,Z 577.786,A -85,B 0,C 180,E1 -17079.849,E2 -17079.849} C_VEL
LIN {X 0,Y 297.777,Z 585.055,A -85,B 0,C 180,E1 -17081.777,E2 -17081.777} C_VEL
LIN {X 0,Y 295.654,Z 590.107,A -85,B 0,C 180,E1 -17083.426,E2 -17083.426} C_VEL
LIN {X 0,Y 293.432,Z 594.889,A -85,B 0,C 180,E1 -17085.435,E2 -17085.435} C_VEL
LIN {X 0,Y 291.401,Z 598.581,A -85,B 0,C 180,E1 -17087.463,E2 -17087.463} C_VEL
LIN {X 0,Y 290.241,Z 600.433,A -85,B 0,C 180,E1 -17088.83,E2 -17088.83} C_VEL
LIN {X 0,Y 289.133,Z 601.848,A -85,B 0,C 180,E1 -17090.203,E2 -17090.203} C_VEL
LIN {X 0,Y 288.111,Z 602.786,A -85,B 0,C 180,E1 -17091.584,E2 -17091.584} C_VEL
LIN {X 0,Y 287.344,Z 603.28,A -85,B 0,C 180,E1 -17092.976,E2 -17092.976} C_VEL
LIN {X 0,Y 286.746,Z 603.371,A -85,B 0,C 180,E1 -17094.374,E2 -17094.374} C_VEL
LIN {X 0,Y 286.21,Z 603.01,A -85,B 0,C 180,E1 -17095.775,E2 -17095.775} C_VEL
LIN {X 0,Y 285.597,Z 602.246,A -85,B 0,C 180,E1 -17097.179,E2 -17097.179} C_VEL
LIN {X 0,Y 285.216,Z 601.049,A -85,B 0,C 180,E1 -17098.588,E2 -17098.588} C_VEL
LIN {X 0,Y 284.715,Z 598.431,A -85,B 0,C 180,E1 -17100.707,E2 -17100.707} C_VEL
LIN {X 0,Y 284.463,Z 594.781,A -85,B 0,C 180,E1 -17102.832,E2 -17102.832} C_VEL
LIN {X 0,Y 284.453,Z 589.988,A -85,B 0,C 180,E1 -17104.961,E2 -17104.961} C_VEL
LIN {X 0,Y 284.736,Z 583.917,A -85,B 0,C 180,E1 -17107.089,E2 -17107.089} C_VEL
LIN {X 0,Y 285.22,Z 575.53,A -85,B 0,C 180,E1 -17109.442,E2 -17109.442} C_VEL
LIN {X 0,Y 285.635,Z 567.153,A -85,B 0,C 180,E1 -17111.352,E2 -17111.352} C_VEL
LIN {X 0,Y 286.319,Z 556.65,A -85,B 0,C 180,E1 -17113.304,E2 -17113.304} C_VEL
LIN {X 0,Y 286.905,Z 546.167,A -85,B 0,C 180,E1 -17114.905,E2 -17114.905} C_VEL
LIN {X 0,Y 287.625,Z 533.091,A -85,B 0,C 180,E1 -17116.502,E2 -17116.502} C_VEL
LIN {X 0,Y 288.264,Z 522,A -85,B 0,C 180,E1 -17117.581,E2 -17117.581} C_VEL
LIN {X 0,Y 288.668,Z 507.876,A -85,B 0,C 180,E1 -17118.636,E2 -17118.636} C_VEL
LIN {X 0,Y 289.024,Z 494.596,A -85,B 0,C 180,E1 -17119.348,E2 -17119.348} C_VEL
LIN {X 0,Y 290.188,Z 446.574,A -85,B 0,C 180,E1 -17121.116,E2 -17121.116} C_VEL
LIN {X 0,Y 290.51,Z 433.905,A -85,B 0,C 180,E1 -17121.584,E2 -17121.584} C_VEL
LIN {X 0,Y 284.578,Z 414.065,A -85,B 0,C 180,E1 -17122.61,E2 -17122.61} C_VEL
LIN {X 0,Y 284.384,Z 413.149,A -85,B 0,C 180,E1 -17122.879,E2 -17122.879} C_VEL
LIN {X 0,Y 284.335,Z 413.059,A -85,B 0,C 180,E1 -17127.149,E2 -17127.149} C_VEL
LIN {X 0,Y 284.3,Z 413.06,A -85,B 0,C 180,E1 -17130.093,E2 -17130.093} C_VEL
LIN {X 0,Y 284.306,Z 413.057,A -85,B 0,C 180,E1 -17132.945,E2 -17132.945} C_VEL
LIN {X 0,Y 284.332,Z 413.069,A -85,B 0,C 180,E1 -17136.386,E2 -17136.386} C_VEL
LIN {X 0,Y 284.307,Z 413.072,A -85,B 0,C 180,E1 -17139.995,E2 -17139.995} C_VEL
LIN {X 0,Y 284.247,Z 413.076,A -85,B 0,C 180,E1 -17144.191,E2 -17144.191} C_VEL
LIN {X 0,Y 284.311,Z 413.255,A -85,B 0,C 180,E1 -17146.364,E2 -17146.364} C_VEL
LIN {X 0,Y 288.365,Z 424.758,A -85,B 0,C 180,E1 -17149.463,E2 -17149.463} C_VEL
LIN {X 0,Y 291.678,Z 435.407,A -85,B 0,C 180,E1 -17152.103,E2 -17152.103} C_VEL
LIN {X 0,Y 294.523,Z 446.228,A -85,B 0,C 180,E1 -17154.62,E2 -17154.62} C_VEL
LIN {X 0,Y 296.913,Z 457.144,A -85,B 0,C 180,E1 -17157.015,E2 -17157.015} C_VEL
LIN {X 0,Y 296.286,Z 464.656,A -85,B 0,C 180,E1 -17158.344,E2 -17158.344} C_VEL
LIN {X 0,Y 293.941,Z 487.992,A -85,B 0,C 180,E1 -17162.265,E2 -17162.265} C_VEL
LIN {X 0,Y 298.677,Z 522.279,A -85,B 0,C 180,E1 -17163.664,E2 -17163.664} C_VEL
LIN {X 0,Y 296.628,Z 598.585,A -85,B 0,C 180,E1 -17165.504,E2 -17165.504} C_VEL
LIN {X 0,Y 295.777,Z 611.898,A -85,B 0,C 180,E1 -17166.036,E2 -17166.036} C_VEL
LIN {X 0,Y 294.662,Z 624.54,A -85,B 0,C 180,E1 -17166.825,E2 -17166.825} C_VEL
LIN {X 0,Y 293.312,Z 636.191,A -85,B 0,C 180,E1 -17167.828,E2 -17167.828} C_VEL
LIN {X 0,Y 291.583,Z 648.201,A -85,B 0,C 180,E1 -17169.175,E2 -17169.175} C_VEL
LIN {X 0,Y 290.033,Z 657.947,A -85,B 0,C 180,E1 -17170.575,E2 -17170.575} C_VEL
LIN {X 0,Y 288.419,Z 667.615,A -85,B 0,C 180,E1 -17172.305,E2 -17172.305} C_VEL
LIN {X 0,Y 286.708,Z 676.848,A -85,B 0,C 180,E1 -17174.357,E2 -17174.357} C_VEL
LIN {X 0,Y 285.241,Z 684.326,A -85,B 0,C 180,E1 -17176.463,E2 -17176.463} C_VEL
LIN {X 0,Y 284.182,Z 690.326,A -85,B 0,C 180,E1 -17178.589,E2 -17178.589} C_VEL
LIN {X 0,Y 283.339,Z 695.073,A -85,B 0,C 180,E1 -17180.722,E2 -17180.722} C_VEL
LIN {X 0,Y 282.819,Z 698.704,A -85,B 0,C 180,E1 -17182.863,E2 -17182.863} C_VEL
LIN {X 0,Y 282.563,Z 700.574,A -85,B 0,C 180,E1 -17184.29,E2 -17184.29} C_VEL
LIN {X 0,Y 282.424,Z 702.001,A -85,B 0,C 180,E1 -17185.719,E2 -17185.719} C_VEL
LIN {X 0,Y 282.364,Z 703,A -85,B 0,C 180,E1 -17187.147,E2 -17187.147} C_VEL
LIN {X 0,Y 282.311,Z 703.617,A -85,B 0,C 180,E1 -17188.574,E2 -17188.574} C_VEL
LIN {X 0,Y 282.296,Z 703.851,A -85,B 0,C 180,E1 -17190,E2 -17190} C_VEL
LIN {X 0,Y 282.311,Z 703.655,A -85,B 0,C 180,E1 -17191.427,E2 -17191.427} C_VEL
LIN {X 0,Y 282.363,Z 703.063,A -85,B 0,C 180,E1 -17192.854,E2 -17192.854} C_VEL
LIN {X 0,Y 282.417,Z 702.088,A -85,B 0,C 180,E1 -17194.282,E2 -17194.282} C_VEL
LIN {X 0,Y 282.559,Z 700.624,A -85,B 0,C 180,E1 -17195.782,E2 -17195.782} C_VEL
LIN {X 0,Y 283.107,Z 696.606,A -85,B 0,C 180,E1 -17198.566,E2 -17198.566} C_VEL
LIN {X 0,Y 283.801,Z 692.307,A -85,B 0,C 180,E1 -17200.704,E2 -17200.704} C_VEL
LIN {X 0,Y 284.818,Z 686.815,A -85,B 0,C 180,E1 -17202.831,E2 -17202.831} C_VEL
LIN {X 0,Y 286.147,Z 679.929,A -85,B 0,C 180,E1 -17204.945,E2 -17204.945} C_VEL
LIN {X 0,Y 287.819,Z 671.317,A -85,B 0,C 180,E1 -17207.039,E2 -17207.039} C_VEL
LIN {X 0,Y 289.475,Z 661.529,A -85,B 0,C 180,E1 -17208.948,E2 -17208.948} C_VEL
LIN {X 0,Y 291.073,Z 651.523,A -85,B 0,C 180,E1 -17210.494,E2 -17210.494} C_VEL
LIN {X 0,Y 292.794,Z 640.485,A -85,B 0,C 180,E1 -17211.842,E2 -17211.842} C_VEL
LIN {X 0,Y 294.225,Z 629.093,A -85,B 0,C 180,E1 -17212.933,E2 -17212.933} C_VEL
LIN {X 0,Y 295.443,Z 616.749,A -85,B 0,C 180,E1 -17213.807,E2 -17213.807} C_VEL
LIN {X 0,Y 296.482,Z 603.035,A -85,B 0,C 180,E1 -17214.462,E2 -17214.462} C_VEL
LIN {X 0,Y 297.191,Z 582.515,A -85,B 0,C 180,E1 -17215.006,E2 -17215.006} C_VEL
LIN {X 0,Y 298.712,Z 522.248,A -85,B 0,C 180,E1 -17216.451,E2 -17216.451} C_VEL
LIN {X 0,Y 294.325,Z 490.309,A -85,B 0,C 180,E1 -17217.737,E2 -17217.737} C_VEL
LIN {X 0,Y 293.983,Z 487.727,A -85,B 0,C 180,E1 -17217.881,E2 -17217.881} C_VEL
LIN {X 0,Y 296.612,Z 462.158,A -85,B 0,C 180,E1 -17222.217,E2 -17222.217} C_VEL
LIN {X 0,Y 297.017,Z 457.922,A -85,B 0,C 180,E1 -17222.972,E2 -17222.972} C_VEL
LIN {X 0,Y 294.774,Z 446.923,A -85,B 0,C 180,E1 -17225.346,E2 -17225.346} C_VEL
LIN {X 0,Y 291.061,Z 432.892,A -85,B 0,C 180,E1 -17228.673,E2 -17228.673} C_VEL
LIN {X 0,Y 290.309,Z 430.605,A -85,B 0,C 180,E1 -17229.229,E2 -17229.229} C_VEL
LIN {X 0,Y 288.598,Z 427.302,A -85,B 0,C 180,E1 -17230.135,E2 -17230.135} C_VEL
LIN {X 0,Y 284.313,Z 422.907,A -85,B 0,C 180,E1 -17231.687,E2 -17231.687} C_VEL
LIN {X 0,Y 278.997,Z 417.853,A -85,B 0,C 180,E1 -17233.62,E2 -17233.62} C_VEL
LIN {X 0,Y 277.716,Z 415.844,A -85,B 0,C 180,E1 -17234.278,E2 -17234.278} C_VEL
LIN {X 0,Y 277.219,Z 414.193,A -85,B 0,C 180,E1 -17234.777,E2 -17234.777} C_VEL
LIN {X 0,Y 277.167,Z 413.929,A -85,B 0,C 180,E1 -17235.234,E2 -17235.234} C_VEL
LIN {X 0,Y 277.187,Z 413.952,A -85,B 0,C 180,E1 -17238.759,E2 -17238.759} C_VEL
LIN {X 0,Y 277.257,Z 413.937,A -85,B 0,C 180,E1 -17242.529,E2 -17242.529} C_VEL
LIN {X 0,Y 277.248,Z 413.936,A -85,B 0,C 180,E1 -17246.104,E2 -17246.104} C_VEL
LIN {X 0,Y 277.23,Z 413.949,A -85,B 0,C 180,E1 -17249.535,E2 -17249.535} C_VEL
LIN {X 0,Y 277.29,Z 413.943,A -85,B 0,C 180,E1 -17252.857,E2 -17252.857} C_VEL
LIN {X 0,Y 277.285,Z 413.926,A -85,B 0,C 180,E1 -17256.075,E2 -17256.075} C_VEL
LIN {X 0,Y 277.282,Z 413.933,A -85,B 0,C 180,E1 -17260.762,E2 -17260.762} C_VEL
LIN {X 0,Y 277.384,Z 413.934,A -85,B 0,C 180,E1 -17265.323,E2 -17265.323} C_VEL
LIN {X 0,Y 277.456,Z 413.902,A -85,B 0,C 180,E1 -17269.787,E2 -17269.787} C_VEL
LIN {X 0,Y 277.603,Z 413.903,A -85,B 0,C 180,E1 -17272.728,E2 -17272.728} C_VEL
LIN {X 0,Y 277.808,Z 413.879,A -85,B 0,C 180,E1 -17278.55,E2 -17278.55} C_VEL
LIN {X 0,Y 277.806,Z 413.855,A -85,B 0,C 180,E1 -17281.45,E2 -17281.45} C_VEL
LIN {X 0,Y 277.604,Z 413.899,A -85,B 0,C 180,E1 -17287.272,E2 -17287.272} C_VEL
LIN {X 0,Y 277.456,Z 413.896,A -85,B 0,C 180,E1 -17290.213,E2 -17290.213} C_VEL
LIN {X 0,Y 277.369,Z 413.925,A -85,B 0,C 180,E1 -17294.678,E2 -17294.678} C_VEL
LIN {X 0,Y 277.271,Z 413.944,A -85,B 0,C 180,E1 -17299.239,E2 -17299.239} C_VEL
LIN {X 0,Y 277.249,Z 413.927,A -85,B 0,C 180,E1 -17302.348,E2 -17302.348} C_VEL
LIN {X 0,Y 277.234,Z 413.949,A -85,B 0,C 180,E1 -17305.528,E2 -17305.528} C_VEL
LIN {X 0,Y 277.219,Z 413.931,A -85,B 0,C 180,E1 -17308.796,E2 -17308.796} C_VEL
LIN {X 0,Y 277.255,Z 413.938,A -85,B 0,C 180,E1 -17313.227,E2 -17313.227} C_VEL
LIN {X 0,Y 277.274,Z 413.938,A -85,B 0,C 180,E1 -17315.796,E2 -17315.796} C_VEL
LIN {X 0,Y 277.217,Z 413.913,A -85,B 0,C 180,E1 -17319.331,E2 -17319.331} C_VEL
LIN {X 0,Y 277.191,Z 413.911,A -85,B 0,C 180,E1 -17323.202,E2 -17323.202} C_VEL
LIN {X 0,Y 277.193,Z 413.922,A -85,B 0,C 180,E1 -17327.33,E2 -17327.33} C_VEL
LIN {X 0,Y 277.292,Z 413.959,A -85,B 0,C 180,E1 -17332.169,E2 -17332.169} C_VEL
LIN {X 0,Y 277.37,Z 414.475,A -85,B 0,C 180,E1 -17332.546,E2 -17332.546} C_VEL
LIN {X 0,Y 278.889,Z 421.631,A -85,B 0,C 180,E1 -17334.381,E2 -17334.381} C_VEL
LIN {X 0,Y 282.439,Z 433.663,A -85,B 0,C 180,E1 -17336.125,E2 -17336.125} C_VEL
LIN {X 0,Y 286.409,Z 446.775,A -85,B 0,C 180,E1 -17337.84,E2 -17337.84} C_VEL
LIN {X 0,Y 287.12,Z 461.753,A -85,B 0,C 180,E1 -17339.231,E2 -17339.231} C_VEL
LIN {X 0,Y 287.469,Z 483.797,A -85,B 0,C 180,E1 -17341.248,E2 -17341.248} C_VEL
LIN {X 0,Y 287.633,Z 489.262,A -85,B 0,C 180,E1 -17341.711,E2 -17341.711} C_VEL
LIN {X 0,Y 291.182,Z 522.605,A -85,B 0,C 180,E1 -17342.993,E2 -17342.993} C_VEL
LIN {X 0,Y 291.712,Z 530.685,A -85,B 0,C 180,E1 -17343.264,E2 -17343.264} C_VEL
LIN {X 0,Y 289.717,Z 602.827,A -85,B 0,C 180,E1 -17345.023,E2 -17345.023} C_VEL
LIN {X 0,Y 288.917,Z 615.661,A -85,B 0,C 180,E1 -17345.525,E2 -17345.525} C_VEL
LIN {X 0,Y 287.81,Z 627.512,A -85,B 0,C 180,E1 -17346.239,E2 -17346.239} C_VEL
LIN {X 0,Y 286.407,Z 639.598,A -85,B 0,C 180,E1 -17347.264,E2 -17347.264} C_VEL
LIN {X 0,Y 284.626,Z 651.907,A -85,B 0,C 180,E1 -17348.641,E2 -17348.641} C_VEL
LIN {X 0,Y 282.784,Z 662.68,A -85,B 0,C 180,E1 -17350.207,E2 -17350.207} C_VEL
LIN {X 0,Y 281.136,Z 672.351,A -85,B 0,C 180,E1 -17351.982,E2 -17351.982} C_VEL
LIN {X 0,Y 279.529,Z 680.962,A -85,B 0,C 180,E1 -17353.944,E2 -17353.944} C_VEL
LIN {X 0,Y 277.981,Z 688.502,A -85,B 0,C 180,E1 -17356.102,E2 -17356.102} C_VEL
LIN {X 0,Y 276.939,Z 694.556,A -85,B 0,C 180,E1 -17358.286,E2 -17358.286} C_VEL
LIN {X 0,Y 276.135,Z 699.335,A -85,B 0,C 180,E1 -17360.477,E2 -17360.477} C_VEL
LIN {X 0,Y 275.622,Z 702.981,A -85,B 0,C 180,E1 -17362.675,E2 -17362.675} C_VEL
LIN {X 0,Y 275.41,Z 705.13,A -85,B 0,C 180,E1 -17364.394,E2 -17364.394} C_VEL
LIN {X 0,Y 275.304,Z 707.275,A -85,B 0,C 180,E1 -17367.073,E2 -17367.073} C_VEL
LIN {X 0,Y 275.285,Z 707.885,A -85,B 0,C 180,E1 -17368.537,E2 -17368.537} C_VEL
LIN {X 0,Y 275.288,Z 708.101,A -85,B 0,C 180,E1 -17370,E2 -17370} C_VEL
LIN {X 0,Y 275.309,Z 707.877,A -85,B 0,C 180,E1 -17371.463,E2 -17371.463} C_VEL
LIN {X 0,Y 275.332,Z 707.262,A -85,B 0,C 180,E1 -17372.926,E2 -17372.926} C_VEL
LIN {X 0,Y 275.416,Z 705.094,A -85,B 0,C 180,E1 -17375.618,E2 -17375.618} C_VEL
LIN {X 0,Y 275.763,Z 701.866,A -85,B 0,C 180,E1 -17378.058,E2 -17378.058} C_VEL
LIN {X 0,Y 276.381,Z 697.84,A -85,B 0,C 180,E1 -17380.253,E2 -17380.253} C_VEL
LIN {X 0,Y 277.421,Z 691.631,A -85,B 0,C 180,E1 -17382.807,E2 -17382.807} C_VEL
LIN {X 0,Y 278.774,Z 684.855,A -85,B 0,C 180,E1 -17384.975,E2 -17384.975} C_VEL
LIN {X 0,Y 280.058,Z 677.918,A -85,B 0,C 180,E1 -17386.773,E2 -17386.773} C_VEL
LIN {X 0,Y 281.678,Z 669.032,A -85,B 0,C 180,E1 -17388.648,E2 -17388.648} C_VEL
LIN {X 0,Y 283.36,Z 659.159,A -85,B 0,C 180,E1 -17390.318,E2 -17390.318} C_VEL
LIN {X 0,Y 285.031,Z 648.881,A -85,B 0,C 180,E1 -17391.707,E2 -17391.707} C_VEL
LIN {X 0,Y 286.615,Z 637.575,A -85,B 0,C 180,E1 -17392.909,E2 -17392.909} C_VEL
LIN {X 0,Y 287.829,Z 627.486,A -85,B 0,C 180,E1 -17393.759,E2 -17393.759} C_VEL
LIN {X 0,Y 291.343,Z 616.926,A -85,B 0,C 180,E1 -17395.352,E2 -17395.352} C_VEL
LIN {X 0,Y 295.277,Z 604.112,A -85,B 0,C 180,E1 -17396.887,E2 -17396.887} C_VEL
LIN {X 0,Y 298.669,Z 591.613,A -85,B 0,C 180,E1 -17398.075,E2 -17398.075} C_VEL
LIN {X 0,Y 302.049,Z 576.921,A -85,B 0,C 180,E1 -17399.155,E2 -17399.155} C_VEL
LIN {X 0,Y 304.923,Z 560.733,A -85,B 0,C 180,E1 -17400.039,E2 -17400.039} C_VEL
LIN {X 0,Y 308.273,Z 532.466,A -85,B 0,C 180,E1 -17401.255,E2 -17401.255} C_VEL
LIN {X 0,Y 309.016,Z 517.268,A -85,B 0,C 180,E1 -17402.199,E2 -17402.199} C_VEL
LIN {X 0,Y 309.006,Z 502.325,A -85,B 0,C 180,E1 -17403.408,E2 -17403.408} C_VEL
LIN {X 0,Y 308.574,Z 488.586,A -85,B 0,C 180,E1 -17404.768,E2 -17404.768} C_VEL
LIN {X 0,Y 307.907,Z 475.354,A -85,B 0,C 180,E1 -17406.356,E2 -17406.356} C_VEL
LIN {X 0,Y 306.846,Z 471.986,A -85,B 0,C 180,E1 -17407.192,E2 -17407.192} C_VEL
LIN {X 0,Y 304.797,Z 465.334,A -85,B 0,C 180,E1 -17409.112,E2 -17409.112} C_VEL
LIN {X 0,Y 302.58,Z 458.912,A -85,B 0,C 180,E1 -17411.889,E2 -17411.889} C_VEL
LIN {X 0,Y 301.681,Z 455.313,A -85,B 0,C 180,E1 -17414.154,E2 -17414.154} C_VEL
LIN {X 0,Y 301.602,Z 453.042,A -85,B 0,C 180,E1 -17416.496,E2 -17416.496} C_VEL
LIN {X 0,Y 302.404,Z 451.855,A -85,B 0,C 180,E1 -17418.676,E2 -17418.676} C_VEL
LIN {X 0,Y 303.754,Z 451.945,A -85,B 0,C 180,E1 -17420.644,E2 -17420.644} C_VEL
LIN {X 0,Y 306.125,Z 453.044,A -85,B 0,C 180,E1 -17422.866,E2 -17422.866} C_VEL
LIN {X 0,Y 309.079,Z 455.725,A -85,B 0,C 180,E1 -17424.944,E2 -17424.944} C_VEL
LIN {X 0,Y 311.874,Z 458.891,A -85,B 0,C 180,E1 -17426.568,E2 -17426.568} C_VEL
LIN {X 0,Y 314.124,Z 463.121,A -85,B 0,C 180,E1 -17427.84,E2 -17427.84} C_VEL
LIN {X 0,Y 315.444,Z 466.021,A -85,B 0,C 180,E1 -17428.54,E2 -17428.54} C_VEL
LIN {X 0,Y 311.383,Z 496.018,A -85,B 0,C 180,E1 -17429.867,E2 -17429.867} C_VEL
LIN {X 0,Y 309.391,Z 515.256,A -85,B 0,C 180,E1 -17430.859,E2 -17430.859} C_VEL
LIN {X 0,Y 307.53,Z 529.576,A -85,B 0,C 180,E1 -17431.878,E2 -17431.878} C_VEL
LIN {X 0,Y 305.71,Z 539.778,A -85,B 0,C 180,E1 -17432.812,E2 -17432.812} C_VEL
LIN {X 0,Y 303.093,Z 552.124,A -85,B 0,C 180,E1 -17434.229,E2 -17434.229} C_VEL
LIN {X 0,Y 300.104,Z 563.117,A -85,B 0,C 180,E1 -17435.806,E2 -17435.806} C_VEL
LIN {X 0,Y 297.168,Z 572.735,A -85,B 0,C 180,E1 -17437.564,E2 -17437.564} C_VEL
LIN {X 0,Y 294.298,Z 580.847,A -85,B 0,C 180,E1 -17439.406,E2 -17439.406} C_VEL
LIN {X 0,Y 291.475,Z 587.746,A -85,B 0,C 180,E1 -17441.368,E2 -17441.368} C_VEL
LIN {X 0,Y 288.452,Z 594.167,A -85,B 0,C 180,E1 -17443.728,E2 -17443.728} C_VEL
LIN {X 0,Y 286.1,Z 598.354,A -85,B 0,C 180,E1 -17445.78,E2 -17445.78} C_VEL
LIN {X 0,Y 284.733,Z 600.51,A -85,B 0,C 180,E1 -17447.165,E2 -17447.165} C_VEL
LIN {X 0,Y 283.505,Z 602.195,A -85,B 0,C 180,E1 -17448.561,E2 -17448.561} C_VEL
LIN {X 0,Y 282.326,Z 603.447,A -85,B 0,C 180,E1 -17449.965,E2 -17449.965} C_VEL
LIN {X 0,Y 281.247,Z 604.282,A -85,B 0,C 180,E1 -17451.377,E2 -17451.377} C_VEL
LIN {X 0,Y 280.435,Z 604.665,A -85,B 0,C 180,E1 -17452.802,E2 -17452.802} C_VEL
LIN {X 0,Y 279.79,Z 604.578,A -85,B 0,C 180,E1 -17454.233,E2 -17454.233} C_VEL
LIN {X 0,Y 279.232,Z 604.082,A -85,B 0,C 180,E1 -17455.67,E2 -17455.67} C_VEL
LIN {X 0,Y 278.588,Z 603.213,A -85,B 0,C 180,E1 -17457.108,E2 -17457.108} C_VEL
LIN {X 0,Y 278.183,Z 601.874,A -85,B 0,C 180,E1 -17458.552,E2 -17458.552} C_VEL
LIN {X 0,Y 277.645,Z 599.05,A -85,B 0,C 180,E1 -17460.725,E2 -17460.725} C_VEL
LIN {X 0,Y 277.382,Z 595.172,A -85,B 0,C 180,E1 -17462.905,E2 -17462.905} C_VEL
LIN {X 0,Y 277.381,Z 590.152,A -85,B 0,C 180,E1 -17465.088,E2 -17465.088} C_VEL
LIN {X 0,Y 277.673,Z 583.868,A -85,B 0,C 180,E1 -17467.27,E2 -17467.27} C_VEL
LIN {X 0,Y 278.127,Z 575.97,A -85,B 0,C 180,E1 -17469.485,E2 -17469.485} C_VEL
LIN {X 0,Y 278.618,Z 566.416,A -85,B 0,C 180,E1 -17471.642,E2 -17471.642} C_VEL
LIN {X 0,Y 279.281,Z 556.599,A -85,B 0,C 180,E1 -17473.46,E2 -17473.46} C_VEL
LIN {X 0,Y 279.872,Z 545.789,A -85,B 0,C 180,E1 -17475.102,E2 -17475.102} C_VEL
LIN {X 0,Y 280.555,Z 534.017,A -85,B 0,C 180,E1 -17476.556,E2 -17476.556} C_VEL
LIN {X 0,Y 281.246,Z 521.222,A -85,B 0,C 180,E1 -17477.809,E2 -17477.809} C_VEL
LIN {X 0,Y 281.636,Z 507.513,A -85,B 0,C 180,E1 -17478.835,E2 -17478.835} C_VEL
LIN {X 0,Y 282.004,Z 493.658,A -85,B 0,C 180,E1 -17479.566,E2 -17479.566} C_VEL
LIN {X 0,Y 283.205,Z 447.15,A -85,B 0,C 180,E1 -17481.348,E2 -17481.348} C_VEL
LIN {X 0,Y 283.529,Z 435.229,A -85,B 0,C 180,E1 -17481.798,E2 -17481.798} C_VEL
LIN {X 0,Y 277.499,Z 414.782,A -85,B 0,C 180,E1 -17482.885,E2 -17482.885} C_VEL
LIN {X 0,Y 277.347,Z 413.993,A -85,B 0,C 180,E1 -17483.177,E2 -17483.177} C_VEL
LIN {X 0,Y 277.275,Z 413.933,A -85,B 0,C 180,E1 -17487.485,E2 -17487.485} C_VEL
LIN {X 0,Y 277.249,Z 413.943,A -85,B 0,C 180,E1 -17490.473,E2 -17490.473} C_VEL
LIN {X 0,Y 277.248,Z 413.931,A -85,B 0,C 180,E1 -17493.896,E2 -17493.896} C_VEL
LIN {X 0,Y 277.266,Z 413.937,A -85,B 0,C 180,E1 -17497.47,E2 -17497.47} C_VEL
LIN {X 0,Y 277.211,Z 413.947,A -85,B 0,C 180,E1 -17501.237,E2 -17501.237} C_VEL
LIN {X 0,Y 277.21,Z 414.109,A -85,B 0,C 180,E1 -17505.322,E2 -17505.322} C_VEL
LIN {X 0,Y 280.803,Z 423.979,A -85,B 0,C 180,E1 -17508.124,E2 -17508.124} C_VEL
LIN {X 0,Y 284.558,Z 435.544,A -85,B 0,C 180,E1 -17511.123,E2 -17511.123} C_VEL
LIN {X 0,Y 287.947,Z 448.143,A -85,B 0,C 180,E1 -17514.142,E2 -17514.142} C_VEL
LIN {X 0,Y 290.353,Z 459.057,A -85,B 0,C 180,E1 -17516.587,E2 -17516.587} C_VEL
LIN {X 0,Y 290.249,Z 462.289,A -85,B 0,C 180,E1 -17517.195,E2 -17517.195} C_VEL
LIN {X 0,Y 287.586,Z 486.595,A -85,B 0,C 180,E1 -17521.382,E2 -17521.382} C_VEL
LIN {X 0,Y 287.567,Z 488.501,A -85,B 0,C 180,E1 -17521.622,E2 -17521.622} C_VEL
LIN {X 0,Y 292.357,Z 523.591,A -85,B 0,C 180,E1 -17523.086,E2 -17523.086} C_VEL
LIN {X 0,Y 290.141,Z 599.896,A -85,B 0,C 180,E1 -17524.967,E2 -17524.967} C_VEL
LIN {X 0,Y 289.263,Z 612.763,A -85,B 0,C 180,E1 -17525.509,E2 -17525.509} C_VEL
LIN {X 0,Y 288.046,Z 625.65,A -85,B 0,C 180,E1 -17526.356,E2 -17526.356} C_VEL
LIN {X 0,Y 286.51,Z 637.933,A -85,B 0,C 180,E1 -17527.463,E2 -17527.463} C_VEL
LIN {X 0,Y 284.961,Z 648.247,A -85,B 0,C 180,E1 -17528.668,E2 -17528.668} C_VEL
LIN {X 0,Y 283.331,Z 657.996,A -85,B 0,C 180,E1 -17530.096,E2 -17530.096} C_VEL
LIN {X 0,Y 281.586,Z 667.949,A -85,B 0,C 180,E1 -17531.922,E2 -17531.922} C_VEL
LIN {X 0,Y 279.875,Z 676.901,A -85,B 0,C 180,E1 -17533.965,E2 -17533.965} C_VEL
LIN {X 0,Y 278.325,Z 684.379,A -85,B 0,C 180,E1 -17536.12,E2 -17536.12} C_VEL
LIN {X 0,Y 277.195,Z 690.38,A -85,B 0,C 180,E1 -17538.298,E2 -17538.298} C_VEL
LIN {X 0,Y 276.328,Z 695.127,A -85,B 0,C 180,E1 -17540.484,E2 -17540.484} C_VEL
LIN {X 0,Y 275.776,Z 698.759,A -85,B 0,C 180,E1 -17542.68,E2 -17542.68} C_VEL
LIN {X 0,Y 275.48,Z 700.752,A -85,B 0,C 180,E1 -17544.248,E2 -17544.248} C_VEL
LIN {X 0,Y 275.277,Z 703.055,A -85,B 0,C 180,E1 -17547.073,E2 -17547.073} C_VEL
LIN {X 0,Y 275.238,Z 703.671,A -85,B 0,C 180,E1 -17548.537,E2 -17548.537} C_VEL
LIN {X 0,Y 275.221,Z 703.905,A -85,B 0,C 180,E1 -17550,E2 -17550} C_VEL
LIN {X 0,Y 275.238,Z 703.708,A -85,B 0,C 180,E1 -17551.463,E2 -17551.463} C_VEL
LIN {X 0,Y 275.276,Z 703.117,A -85,B 0,C 180,E1 -17552.927,E2 -17552.927} C_VEL
LIN {X 0,Y 275.485,Z 700.868,A -85,B 0,C 180,E1 -17555.761,E2 -17555.761} C_VEL
LIN {X 0,Y 275.882,Z 697.871,A -85,B 0,C 180,E1 -17558.054,E2 -17558.054} C_VEL
LIN {X 0,Y 276.544,Z 693.939,A -85,B 0,C 180,E1 -17560.247,E2 -17560.247} C_VEL
LIN {X 0,Y 277.494,Z 688.846,A -85,B 0,C 180,E1 -17562.432,E2 -17562.432} C_VEL
LIN {X 0,Y 278.73,Z 682.426,A -85,B 0,C 180,E1 -17564.605,E2 -17564.605} C_VEL
LIN {X 0,Y 280.449,Z 674.45,A -85,B 0,C 180,E1 -17566.75,E2 -17566.75} C_VEL
LIN {X 0,Y 281.936,Z 666.397,A -85,B 0,C 180,E1 -17568.51,E2 -17568.51} C_VEL
LIN {X 0,Y 283.615,Z 656.26,A -85,B 0,C 180,E1 -17570.299,E2 -17570.299} C_VEL
LIN {X 0,Y 285.532,Z 644.973,A -85,B 0,C 180,E1 -17571.857,E2 -17571.857} C_VEL
LIN {X 0,Y 287.151,Z 633.875,A -85,B 0,C 180,E1 -17573.054,E2 -17573.054} C_VEL
LIN {X 0,Y 288.538,Z 621.306,A -85,B 0,C 180,E1 -17574.079,E2 -17574.079} C_VEL
LIN {X 0,Y 289.735,Z 608.107,A -85,B 0,C 180,E1 -17574.831,E2 -17574.831} C_VEL
LIN {X 0,Y 290.448,Z 594.818,A -85,B 0,C 180,E1 -17575.292,E2 -17575.292} C_VEL
LIN {X 0,Y 292.351,Z 523.09,A -85,B 0,C 180,E1 -17577.048,E2 -17577.048} C_VEL
LIN {X 0,Y 288.069,Z 491.509,A -85,B 0,C 180,E1 -17578.358,E2 -17578.358} C_VEL
LIN {X 0,Y 287.527,Z 487.868,A -85,B 0,C 180,E1 -17578.544,E2 -17578.544} C_VEL
LIN {X 0,Y 290.108,Z 464.127,A -85,B 0,C 180,E1 -17582.617,E2 -17582.617} C_VEL
LIN {X 0,Y 290.495,Z 459.838,A -85,B 0,C 180,E1 -17583.395,E2 -17583.395} C_VEL
LIN {X 0,Y 288.156,Z 448.793,A -85,B 0,C 180,E1 -17585.828,E2 -17585.828} C_VEL
LIN {X 0,Y 284.744,Z 435.832,A -85,B 0,C 180,E1 -17588.969,E2 -17588.969} C_VEL
LIN {X 0,Y 280.973,Z 424.458,A -85,B 0,C 180,E1 -17591.915,E2 -17591.915} C_VEL
LIN {X 0,Y 277.716,Z 415.844,A -85,B 0,C 180,E1 -17594.278,E2 -17594.278} C_VEL
LIN {X 0,Y 276.572,Z 414.516,A -85,B 0,C 180,E1 -17594.966,E2 -17594.966} C_VEL
LIN {X 0,Y 274.65,Z 414.25,A -85,B 0,C 180,E1 -17596.103,E2 -17596.103} C_VEL
LIN {X 0,Y 270.885,Z 414.832,A -85,B 0,C 180,E1 -17598.963,E2 -17598.963} C_VEL
LIN {X 0,Y 270.153,Z 414.827,A -85,B 0,C 180,E1 -17600.688,E2 -17600.688} C_VEL
LIN {X 0,Y 270.222,Z 414.818,A -85,B 0,C 180,E1 -17603.733,E2 -17603.733} C_VEL
LIN {X 0,Y 270.204,Z 414.812,A -85,B 0,C 180,E1 -17606.892,E2 -17606.892} C_VEL
LIN {X 0,Y 270.161,Z 414.82,A -85,B 0,C 180,E1 -17610.378,E2 -17610.378} C_VEL
LIN {X 0,Y 270.202,Z 414.831,A -85,B 0,C 180,E1 -17613.757,E2 -17613.757} C_VEL
LIN {X 0,Y 270.201,Z 414.809,A -85,B 0,C 180,E1 -17617.036,E2 -17617.036} C_VEL
LIN {X 0,Y 270.224,Z 414.82,A -85,B 0,C 180,E1 -17620.238,E2 -17620.238} C_VEL
LIN {X 0,Y 270.347,Z 414.809,A -85,B 0,C 180,E1 -17624.932,E2 -17624.932} C_VEL
LIN {X 0,Y 270.388,Z 414.779,A -85,B 0,C 180,E1 -17629.517,E2 -17629.517} C_VEL
LIN {X 0,Y 270.565,Z 414.78,A -85,B 0,C 180,E1 -17632.537,E2 -17632.537} C_VEL
LIN {X 0,Y 270.773,Z 414.755,A -85,B 0,C 180,E1 -17638.513,E2 -17638.513} C_VEL
LIN {X 0,Y 270.771,Z 414.73,A -85,B 0,C 180,E1 -17641.487,E2 -17641.487} C_VEL
LIN {X 0,Y 270.565,Z 414.773,A -85,B 0,C 180,E1 -17647.462,E2 -17647.462} C_VEL
LIN {X 0,Y 270.389,Z 414.777,A -85,B 0,C 180,E1 -17650.483,E2 -17650.483} C_VEL
LIN {X 0,Y 270.34,Z 414.792,A -85,B 0,C 180,E1 -17655.068,E2 -17655.068} C_VEL
LIN {X 0,Y 270.218,Z 414.827,A -85,B 0,C 180,E1 -17659.762,E2 -17659.762} C_VEL
LIN {X 0,Y 270.184,Z 414.813,A -85,B 0,C 180,E1 -17664.436,E2 -17664.436} C_VEL
LIN {X 0,Y 270.186,Z 414.813,A -85,B 0,C 180,E1 -17667.918,E2 -17667.918} C_VEL
LIN {X 0,Y 270.171,Z 414.83,A -85,B 0,C 180,E1 -17671.35,E2 -17671.35} C_VEL
LIN {X 0,Y 270.199,Z 414.81,A -85,B 0,C 180,E1 -17674.906,E2 -17674.906} C_VEL
LIN {X 0,Y 270.2,Z 414.8,A -85,B 0,C 180,E1 -17678.71,E2 -17678.71} C_VEL
LIN {X 0,Y 270.149,Z 414.787,A -85,B 0,C 180,E1 -17683.244,E2 -17683.244} C_VEL
LIN {X 0,Y 270.152,Z 414.796,A -85,B 0,C 180,E1 -17687.437,E2 -17687.437} C_VEL
LIN {X 0,Y 270.261,Z 415.021,A -85,B 0,C 180,E1 -17692.062,E2 -17692.062} C_VEL
LIN {X 0,Y 270.527,Z 416.171,A -85,B 0,C 180,E1 -17692.405,E2 -17692.405} C_VEL
LIN {X 0,Y 276.095,Z 434.264,A -85,B 0,C 180,E1 -17695.191,E2 -17695.191} C_VEL
LIN {X 0,Y 280.484,Z 449.451,A -85,B 0,C 180,E1 -17697.247,E2 -17697.247} C_VEL
LIN {X 0,Y 281.101,Z 469.292,A -85,B 0,C 180,E1 -17699.145,E2 -17699.145} C_VEL
LIN {X 0,Y 281.248,Z 488.997,A -85,B 0,C 180,E1 -17700.998,E2 -17700.998} C_VEL
LIN {X 0,Y 284.88,Z 523.43,A -85,B 0,C 180,E1 -17702.365,E2 -17702.365} C_VEL
LIN {X 0,Y 285.375,Z 532.593,A -85,B 0,C 180,E1 -17702.671,E2 -17702.671} C_VEL
LIN {X 0,Y 283.307,Z 602.876,A -85,B 0,C 180,E1 -17704.418,E2 -17704.418} C_VEL
LIN {X 0,Y 282.487,Z 615.665,A -85,B 0,C 180,E1 -17704.93,E2 -17704.93} C_VEL
LIN {X 0,Y 281.321,Z 627.492,A -85,B 0,C 180,E1 -17705.656,E2 -17705.656} C_VEL
LIN {X 0,Y 279.865,Z 639.568,A -85,B 0,C 180,E1 -17706.702,E2 -17706.702} C_VEL
LIN {X 0,Y 278.022,Z 651.869,A -85,B 0,C 180,E1 -17708.108,E2 -17708.108} C_VEL
LIN {X 0,Y 276.097,Z 662.637,A -85,B 0,C 180,E1 -17709.707,E2 -17709.707} C_VEL
LIN {X 0,Y 274.252,Z 672.974,A -85,B 0,C 180,E1 -17711.66,E2 -17711.66} C_VEL
LIN {X 0,Y 272.687,Z 680.914,A -85,B 0,C 180,E1 -17713.53,E2 -17713.53} C_VEL
LIN {X 0,Y 271.081,Z 688.452,A -85,B 0,C 180,E1 -17715.741,E2 -17715.741} C_VEL
LIN {X 0,Y 269.957,Z 694.505,A -85,B 0,C 180,E1 -17717.979,E2 -17717.979} C_VEL
LIN {X 0,Y 269.104,Z 699.282,A -85,B 0,C 180,E1 -17720.226,E2 -17720.226} C_VEL
LIN {X 0,Y 268.553,Z 702.928,A -85,B 0,C 180,E1 -17722.481,E2 -17722.481} C_VEL
LIN {X 0,Y 268.324,Z 705.271,A -85,B 0,C 180,E1 -17724.448,E2 -17724.448} C_VEL
LIN {X 0,Y 268.217,Z 707.222,A -85,B 0,C 180,E1 -17726.996,E2 -17726.996} C_VEL
LIN {X 0,Y 268.211,Z 707.832,A -85,B 0,C 180,E1 -17728.498,E2 -17728.498} C_VEL
LIN {X 0,Y 268.212,Z 708.047,A -85,B 0,C 180,E1 -17730,E2 -17730} C_VEL
LIN {X 0,Y 268.234,Z 707.823,A -85,B 0,C 180,E1 -17731.501,E2 -17731.501} C_VEL
LIN {X 0,Y 268.244,Z 707.208,A -85,B 0,C 180,E1 -17733.003,E2 -17733.003} C_VEL
LIN {X 0,Y 268.333,Z 705.226,A -85,B 0,C 180,E1 -17735.573,E2 -17735.573} C_VEL
LIN {X 0,Y 268.715,Z 701.811,A -85,B 0,C 180,E1 -17738.27,E2 -17738.27} C_VEL
LIN {X 0,Y 269.362,Z 697.786,A -85,B 0,C 180,E1 -17740.523,E2 -17740.523} C_VEL
LIN {X 0,Y 270.455,Z 691.577,A -85,B 0,C 180,E1 -17743.143,E2 -17743.143} C_VEL
LIN {X 0,Y 271.889,Z 684.802,A -85,B 0,C 180,E1 -17745.364,E2 -17745.364} C_VEL
LIN {X 0,Y 273.222,Z 677.866,A -85,B 0,C 180,E1 -17747.206,E2 -17747.206} C_VEL
LIN {X 0,Y 274.879,Z 669.331,A -85,B 0,C 180,E1 -17749.057,E2 -17749.057} C_VEL
LIN {X 0,Y 276.701,Z 659.111,A -85,B 0,C 180,E1 -17750.829,E2 -17750.829} C_VEL
LIN {X 0,Y 278.448,Z 648.836,A -85,B 0,C 180,E1 -17752.247,E2 -17752.247} C_VEL
LIN {X 0,Y 280.097,Z 637.535,A -85,B 0,C 180,E1 -17753.473,E2 -17753.473} C_VEL
LIN {X 0,Y 281.095,Z 629.658,A -85,B 0,C 180,E1 -17754.168,E2 -17754.168} C_VEL
LIN {X 0,Y 285.019,Z 618.745,A -85,B 0,C 180,E1 -17755.956,E2 -17755.956} C_VEL
LIN {X 0,Y 289.492,Z 605.487,A -85,B 0,C 180,E1 -17757.665,E2 -17757.665} C_VEL
LIN {X 0,Y 293.944,Z 590.379,A -85,B 0,C 180,E1 -17759.154,E2 -17759.154} C_VEL
LIN {X 0,Y 297.279,Z 576.962,A -85,B 0,C 180,E1 -17760.157,E2 -17760.157} C_VEL
LIN {X 0,Y 300.292,Z 561.777,A -85,B 0,C 180,E1 -17761.036,E2 -17761.036} C_VEL
LIN {X 0,Y 304.045,Z 533.216,A -85,B 0,C 180,E1 -17762.314,E2 -17762.314} C_VEL
LIN {X 0,Y 304.917,Z 519.096,A -85,B 0,C 180,E1 -17763.221,E2 -17763.221} C_VEL
LIN {X 0,Y 305.142,Z 504.264,A -85,B 0,C 180,E1 -17764.467,E2 -17764.467} C_VEL
LIN {X 0,Y 304.975,Z 490.274,A -85,B 0,C 180,E1 -17765.923,E2 -17765.923} C_VEL
LIN {X 0,Y 304.676,Z 479.787,A -85,B 0,C 180,E1 -17767.231,E2 -17767.231} C_VEL
LIN {X 0,Y 302.34,Z 471.411,A -85,B 0,C 180,E1 -17769.627,E2 -17769.627} C_VEL
LIN {X 0,Y 300.421,Z 464.971,A -85,B 0,C 180,E1 -17772.497,E2 -17772.497} C_VEL
LIN {X 0,Y 299.807,Z 461.687,A -85,B 0,C 180,E1 -17774.689,E2 -17774.689} C_VEL
LIN {X 0,Y 299.994,Z 459.504,A -85,B 0,C 180,E1 -17777.204,E2 -17777.204} C_VEL
LIN {X 0,Y 300.9,Z 458.685,A -85,B 0,C 180,E1 -17779.157,E2 -17779.157} C_VEL
LIN {X 0,Y 302.398,Z 459.056,A -85,B 0,C 180,E1 -17781.134,E2 -17781.134} C_VEL
LIN {X 0,Y 304.161,Z 459.85,A -85,B 0,C 180,E1 -17782.744,E2 -17782.744} C_VEL
LIN {X 0,Y 306.785,Z 462.295,A -85,B 0,C 180,E1 -17784.68,E2 -17784.68} C_VEL
LIN {X 0,Y 309.338,Z 465.245,A -85,B 0,C 180,E1 -17786.237,E2 -17786.237} C_VEL
LIN {X 0,Y 311.475,Z 469.729,A -85,B 0,C 180,E1 -17787.53,E2 -17787.53} C_VEL
LIN {X 0,Y 306.95,Z 501.571,A -85,B 0,C 180,E1 -17788.996,E2 -17788.996} C_VEL
LIN {X 0,Y 305.144,Z 517.765,A -85,B 0,C 180,E1 -17789.89,E2 -17789.89} C_VEL
LIN {X 0,Y 303.175,Z 531.058,A -85,B 0,C 180,E1 -17790.869,E2 -17790.869} C_VEL
LIN {X 0,Y 301.243,Z 541.293,A -85,B 0,C 180,E1 -17791.808,E2 -17791.808} C_VEL
LIN {X 0,Y 298.424,Z 553.428,A -85,B 0,C 180,E1 -17793.231,E2 -17793.231} C_VEL
LIN {X 0,Y 295.566,Z 563.335,A -85,B 0,C 180,E1 -17794.659,E2 -17794.659} C_VEL
LIN {X 0,Y 292.59,Z 572.441,A -85,B 0,C 180,E1 -17796.276,E2 -17796.276} C_VEL
LIN {X 0,Y 289.484,Z 580.802,A -85,B 0,C 180,E1 -17798.137,E2 -17798.137} C_VEL
LIN {X 0,Y 286.192,Z 588.414,A -85,B 0,C 180,E1 -17800.266,E2 -17800.266} C_VEL
LIN {X 0,Y 282.852,Z 594.998,A -85,B 0,C 180,E1 -17802.653,E2 -17802.653} C_VEL
LIN {X 0,Y 279.522,Z 600.434,A -85,B 0,C 180,E1 -17805.438,E2 -17805.438} C_VEL
LIN {X 0,Y 278.077,Z 602.439,A -85,B 0,C 180,E1 -17806.852,E2 -17806.852} C_VEL
LIN {X 0,Y 276.78,Z 603.956,A -85,B 0,C 180,E1 -17808.28,E2 -17808.28} C_VEL
LIN {X 0,Y 275.533,Z 605.068,A -85,B 0,C 180,E1 -17809.715,E2 -17809.715} C_VEL
LIN {X 0,Y 274.398,Z 605.752,A -85,B 0,C 180,E1 -17811.16,E2 -17811.16} C_VEL
LIN {X 0,Y 273.513,Z 605.967,A -85,B 0,C 180,E1 -17812.618,E2 -17812.618} C_VEL
LIN {X 0,Y 272.832,Z 605.762,A -85,B 0,C 180,E1 -17814.086,E2 -17814.086} C_VEL
LIN {X 0,Y 272.25,Z 605.152,A -85,B 0,C 180,E1 -17815.558,E2 -17815.558} C_VEL
LIN {X 0,Y 271.578,Z 604.115,A -85,B 0,C 180,E1 -17817.033,E2 -17817.033} C_VEL
LIN {X 0,Y 271.124,Z 602.638,A -85,B 0,C 180,E1 -17818.515,E2 -17818.515} C_VEL
LIN {X 0,Y 270.577,Z 599.612,A -85,B 0,C 180,E1 -17820.744,E2 -17820.744} C_VEL
LIN {X 0,Y 270.303,Z 595.513,A -85,B 0,C 180,E1 -17822.981,E2 -17822.981} C_VEL
LIN {X 0,Y 270.363,Z 589.263,A -85,B 0,C 180,E1 -17825.594,E2 -17825.594} C_VEL
LIN {X 0,Y 270.749,Z 581.689,A -85,B 0,C 180,E1 -17828.056,E2 -17828.056} C_VEL
LIN {X 0,Y 271.193,Z 573.618,A -85,B 0,C 180,E1 -17830.189,E2 -17830.189} C_VEL
LIN {X 0,Y 271.754,Z 563.705,A -85,B 0,C 180,E1 -17832.319,E2 -17832.319} C_VEL
LIN {X 0,Y 272.423,Z 553.052,A -85,B 0,C 180,E1 -17834.187,E2 -17834.187} C_VEL
LIN {X 0,Y 273.117,Z 541.148,A -85,B 0,C 180,E1 -17835.867,E2 -17835.867} C_VEL
LIN {X 0,Y 273.877,Z 527.915,A -85,B 0,C 180,E1 -17837.356,E2 -17837.356} C_VEL
LIN {X 0,Y 274.358,Z 515.486,A -85,B 0,C 180,E1 -17838.443,E2 -17838.443} C_VEL
LIN {X 0,Y 274.791,Z 501.641,A -85,B 0,C 180,E1 -17839.35,E2 -17839.35} C_VEL
LIN {X 0,Y 275.227,Z 480.391,A -85,B 0,C 180,E1 -17840.263,E2 -17840.263} C_VEL
LIN {X 0,Y 276.512,Z 436.364,A -85,B 0,C 180,E1 -17842.004,E2 -17842.004} C_VEL
LIN {X 0,Y 270.465,Z 415.715,A -85,B 0,C 180,E1 -17843.13,E2 -17843.13} C_VEL
LIN {X 0,Y 270.28,Z 414.894,A -85,B 0,C 180,E1 -17843.413,E2 -17843.413} C_VEL
LIN {X 0,Y 270.204,Z 414.808,A -85,B 0,C 180,E1 -17847.916,E2 -17847.916} C_VEL
LIN {X 0,Y 270.175,Z 414.832,A -85,B 0,C 180,E1 -17851.35,E2 -17851.35} C_VEL
LIN {X 0,Y 270.203,Z 414.813,A -85,B 0,C 180,E1 -17854.906,E2 -17854.906} C_VEL
LIN {X 0,Y 270.199,Z 414.815,A -85,B 0,C 180,E1 -17858.71,E2 -17858.71} C_VEL
LIN {X 0,Y 270.167,Z 414.828,A -85,B 0,C 180,E1 -17863.249,E2 -17863.249} C_VEL
LIN {X 0,Y 270.215,Z 415.169,A -85,B 0,C 180,E1 -17864.325,E2 -17864.325} C_VEL
LIN {X 0,Y 274.512,Z 426.701,A -85,B 0,C 180,E1 -17867.667,E2 -17867.667} C_VEL
LIN {X 0,Y 278.382,Z 438.755,A -85,B 0,C 180,E1 -17870.865,E2 -17870.865} C_VEL
LIN {X 0,Y 281.397,Z 450.14,A -85,B 0,C 180,E1 -17873.655,E2 -17873.655} C_VEL
LIN {X 0,Y 283.8,Z 461.038,A -85,B 0,C 180,E1 -17876.149,E2 -17876.149} C_VEL
LIN {X 0,Y 283.881,Z 463.216,A -85,B 0,C 180,E1 -17876.581,E2 -17876.581} C_VEL
LIN {X 0,Y 281.271,Z 485.491,A -85,B 0,C 180,E1 -17880.493,E2 -17880.493} C_VEL
LIN {X 0,Y 281.142,Z 488.504,A -85,B 0,C 180,E1 -17880.913,E2 -17880.913} C_VEL
LIN {X 0,Y 286.023,Z 524.356,A -85,B 0,C 180,E1 -17882.463,E2 -17882.463} C_VEL
LIN {X 0,Y 283.745,Z 599.888,A -85,B 0,C 180,E1 -17884.362,E2 -17884.362} C_VEL
LIN {X 0,Y 282.815,Z 612.784,A -85,B 0,C 180,E1 -17884.912,E2 -17884.912} C_VEL
LIN {X 0,Y 281.561,Z 625.685,A -85,B 0,C 180,E1 -17885.777,E2 -17885.777} C_VEL
LIN {X 0,Y 279.966,Z 637.975,A -85,B 0,C 180,E1 -17886.906,E2 -17886.906} C_VEL
LIN {X 0,Y 278.367,Z 648.293,A -85,B 0,C 180,E1 -17888.137,E2 -17888.137} C_VEL
LIN {X 0,Y 276.505,Z 658.878,A -85,B 0,C 180,E1 -17889.738,E2 -17889.738} C_VEL
LIN {X 0,Y 274.771,Z 668.29,A -85,B 0,C 180,E1 -17891.522,E2 -17891.522} C_VEL
LIN {X 0,Y 273.06,Z 676.953,A -85,B 0,C 180,E1 -17893.554,E2 -17893.554} C_VEL
LIN {X 0,Y 271.43,Z 684.433,A -85,B 0,C 180,E1 -17895.76,E2 -17895.76} C_VEL
LIN {X 0,Y 270.223,Z 690.434,A -85,B 0,C 180,E1 -17897.991,E2 -17897.991} C_VEL
LIN {X 0,Y 269.302,Z 695.181,A -85,B 0,C 180,E1 -17900.234,E2 -17900.234} C_VEL
LIN {X 0,Y 268.731,Z 698.813,A -85,B 0,C 180,E1 -17902.486,E2 -17902.486} C_VEL
LIN {X 0,Y 268.361,Z 701.08,A -85,B 0,C 180,E1 -17904.368,E2 -17904.368} C_VEL
LIN {X 0,Y 268.193,Z 703.109,A -85,B 0,C 180,E1 -17906.996,E2 -17906.996} C_VEL
LIN {X 0,Y 268.145,Z 703.725,A -85,B 0,C 180,E1 -17908.498,E2 -17908.498} C_VEL
LIN {X 0,Y 268.147,Z 703.959,A -85,B 0,C 180,E1 -17910,E2 -17910} C_VEL
LIN {X 0,Y 268.145,Z 703.762,A -85,B 0,C 180,E1 -17911.502,E2 -17911.502} C_VEL
LIN {X 0,Y 268.191,Z 703.17,A -85,B 0,C 180,E1 -17913.004,E2 -17913.004} C_VEL
LIN {X 0,Y 268.363,Z 701.186,A -85,B 0,C 180,E1 -17915.636,E2 -17915.636} C_VEL
LIN {X 0,Y 268.834,Z 697.923,A -85,B 0,C 180,E1 -17918.267,E2 -17918.267} C_VEL
LIN {X 0,Y 269.539,Z 693.991,A -85,B 0,C 180,E1 -17920.517,E2 -17920.517} C_VEL
LIN {X 0,Y 270.552,Z 688.896,A -85,B 0,C 180,E1 -17922.756,E2 -17922.756} C_VEL
LIN {X 0,Y 271.866,Z 682.475,A -85,B 0,C 180,E1 -17924.982,E2 -17924.982} C_VEL
LIN {X 0,Y 273.649,Z 674.497,A -85,B 0,C 180,E1 -17927.179,E2 -17927.179} C_VEL
LIN {X 0,Y 275.337,Z 665.416,A -85,B 0,C 180,E1 -17929.19,E2 -17929.19} C_VEL
LIN {X 0,Y 277.171,Z 655.159,A -85,B 0,C 180,E1 -17930.987,E2 -17930.987} C_VEL
LIN {X 0,Y 278.95,Z 645.01,A -85,B 0,C 180,E1 -17932.4,E2 -17932.4} C_VEL
LIN {X 0,Y 280.629,Z 633.903,A -85,B 0,C 180,E1 -17933.622,E2 -17933.622} C_VEL
LIN {X 0,Y 282.058,Z 621.323,A -85,B 0,C 180,E1 -17934.668,E2 -17934.668} C_VEL
LIN {X 0,Y 283.3,Z 608.099,A -85,B 0,C 180,E1 -17935.435,E2 -17935.435} C_VEL
LIN {X 0,Y 284.051,Z 594.748,A -85,B 0,C 180,E1 -17935.904,E2 -17935.904} C_VEL
LIN {X 0,Y 285.974,Z 523.506,A -85,B 0,C 180,E1 -17937.688,E2 -17937.688} C_VEL
LIN {X 0,Y 281.639,Z 491.377,A -85,B 0,C 180,E1 -17939.067,E2 -17939.067} C_VEL
LIN {X 0,Y 281.114,Z 487.724,A -85,B 0,C 180,E1 -17939.274,E2 -17939.274} C_VEL
LIN {X 0,Y 283.842,Z 463.9,A -85,B 0,C 180,E1 -17943.43,E2 -17943.43} C_VEL
LIN {X 0,Y 283.787,Z 460.668,A -85,B 0,C 180,E1 -17944.078,E2 -17944.078} C_VEL
LIN {X 0,Y 281.553,Z 450.521,A -85,B 0,C 180,E1 -17946.388,E2 -17946.388} C_VEL
LIN {X 0,Y 278.672,Z 439.525,A -85,B 0,C 180,E1 -17949.087,E2 -17949.087} C_VEL
LIN {X 0,Y 274.957,Z 427.983,A -85,B 0,C 180,E1 -17952.162,E2 -17952.162} C_VEL
LIN {X 0,Y 271.249,Z 417.965,A -85,B 0,C 180,E1 -17954.961,E2 -17954.961} C_VEL
LIN {X 0,Y 270.135,Z 414.975,A -85,B 0,C 180,E1 -17955.942,E2 -17955.942} C_VEL
LIN {X 0,Y 270.15,Z 414.827,A -85,B 0,C 180,E1 -17959.429,E2 -17959.429} C_VEL
LIN {X 0,Y 270.153,Z 414.827,A -85,B 0,C 180,E1 -17960.688,E2 -17960.688} C_VEL
LIN {X 0,Y 269.53,Z 414.91,A -85,B 0,C 180,E1 -17961.931,E2 -17961.931} C_VEL
LIN {X 0,Y 266.665,Z 415.264,A -85,B 0,C 180,E1 -17963.957,E2 -17963.957} C_VEL
LIN {X 0,Y 264.216,Z 415.563,A -85,B 0,C 180,E1 -17965.604,E2 -17965.604} C_VEL
LIN {X 0,Y 263.184,Z 415.687,A -85,B 0,C 180,E1 -17966.882,E2 -17966.882} C_VEL
LIN {X 0,Y 263.111,Z 415.698,A -85,B 0,C 180,E1 -17967.315,E2 -17967.315} C_VEL
LIN {X 0,Y 263.144,Z 415.692,A -85,B 0,C 180,E1 -17971.808,E2 -17971.808} C_VEL
LIN {X 0,Y 263.192,Z 415.687,A -85,B 0,C 180,E1 -17975.218,E2 -17975.218} C_VEL
LIN {X 0,Y 263.211,Z 415.698,A -85,B 0,C 180,E1 -17979.689,E2 -17979.689} C_VEL
LIN {X 0,Y 263.293,Z 415.685,A -85,B 0,C 180,E1 -17984.518,E2 -17984.518} C_VEL
LIN {X 0,Y 263.333,Z 415.655,A -85,B 0,C 180,E1 -17989.233,E2 -17989.233} C_VEL
LIN {X 0,Y 263.529,Z 415.657,A -85,B 0,C 180,E1 -17992.337,E2 -17992.337} C_VEL
LIN {X 0,Y 263.736,Z 415.632,A -85,B 0,C 180,E1 -17998.473,E2 -17998.473} C_VEL
LIN {X 0,Y 263.735,Z 415.605,A -85,B 0,C 180,E1 -18001.527,E2 -18001.527} C_VEL
LIN {X 0,Y 263.529,Z 415.646,A -85,B 0,C 180,E1 -18007.663,E2 -18007.663} C_VEL
LIN {X 0,Y 263.334,Z 415.658,A -85,B 0,C 180,E1 -18010.767,E2 -18010.767} C_VEL
LIN {X 0,Y 263.291,Z 415.664,A -85,B 0,C 180,E1 -18015.482,E2 -18015.482} C_VEL
LIN {X 0,Y 263.208,Z 415.698,A -85,B 0,C 180,E1 -18020.311,E2 -18020.311} C_VEL
LIN {X 0,Y 263.122,Z 415.705,A -85,B 0,C 180,E1 -18025.3,E2 -18025.3} C_VEL
LIN {X 0,Y 263.12,Z 415.687,A -85,B 0,C 180,E1 -18028.737,E2 -18028.737} C_VEL
LIN {X 0,Y 263.128,Z 415.707,A -85,B 0,C 180,E1 -18032.289,E2 -18032.289} C_VEL
LIN {X 0,Y 263.158,Z 415.698,A -85,B 0,C 180,E1 -18035.983,E2 -18035.983} C_VEL
LIN {X 0,Y 263.092,Z 415.658,A -85,B 0,C 180,E1 -18039.875,E2 -18039.875} C_VEL
LIN {X 0,Y 263.082,Z 415.682,A -85,B 0,C 180,E1 -18043.993,E2 -18043.993} C_VEL
LIN {X 0,Y 263.076,Z 415.669,A -85,B 0,C 180,E1 -18048.097,E2 -18048.097} C_VEL
LIN {X 0,Y 263.123,Z 415.872,A -85,B 0,C 180,E1 -18050.768,E2 -18050.768} C_VEL
LIN {X 0,Y 263.28,Z 416.513,A -85,B 0,C 180,E1 -18051.033,E2 -18051.033} C_VEL
LIN {X 0,Y 265.391,Z 420.912,A -85,B 0,C 180,E1 -18051.991,E2 -18051.991} C_VEL
LIN {X 0,Y 270.866,Z 439.078,A -85,B 0,C 180,E1 -18054.818,E2 -18054.818} C_VEL
LIN {X 0,Y 274.537,Z 452.12,A -85,B 0,C 180,E1 -18056.652,E2 -18056.652} C_VEL
LIN {X 0,Y 274.978,Z 475.736,A -85,B 0,C 180,E1 -18058.98,E2 -18058.98} C_VEL
LIN {X 0,Y 274.92,Z 488.743,A -85,B 0,C 180,E1 -18060.253,E2 -18060.253} C_VEL
LIN {X 0,Y 278.503,Z 522.872,A -85,B 0,C 180,E1 -18061.658,E2 -18061.658} C_VEL
LIN {X 0,Y 279.095,Z 532.453,A -85,B 0,C 180,E1 -18061.997,E2 -18061.997} C_VEL
LIN {X 0,Y 276.929,Z 602.923,A -85,B 0,C 180,E1 -18063.785,E2 -18063.785} C_VEL
LIN {X 0,Y 276.094,Z 615.668,A -85,B 0,C 180,E1 -18064.308,E2 -18064.308} C_VEL
LIN {X 0,Y 274.877,Z 627.473,A -85,B 0,C 180,E1 -18065.047,E2 -18065.047} C_VEL
LIN {X 0,Y 273.365,Z 639.537,A -85,B 0,C 180,E1 -18066.113,E2 -18066.113} C_VEL
LIN {X 0,Y 271.43,Z 651.832,A -85,B 0,C 180,E1 -18067.547,E2 -18067.547} C_VEL
LIN {X 0,Y 269.438,Z 662.595,A -85,B 0,C 180,E1 -18069.182,E2 -18069.182} C_VEL
LIN {X 0,Y 267.657,Z 671.884,A -85,B 0,C 180,E1 -18070.956,E2 -18070.956} C_VEL
LIN {X 0,Y 265.855,Z 680.866,A -85,B 0,C 180,E1 -18073.094,E2 -18073.094} C_VEL
LIN {X 0,Y 264.199,Z 688.402,A -85,B 0,C 180,E1 -18075.362,E2 -18075.362} C_VEL
LIN {X 0,Y 262.991,Z 694.454,A -85,B 0,C 180,E1 -18077.655,E2 -18077.655} C_VEL
LIN {X 0,Y 262.088,Z 699.23,A -85,B 0,C 180,E1 -18079.962,E2 -18079.962} C_VEL
LIN {X 0,Y 261.512,Z 702.876,A -85,B 0,C 180,E1 -18082.277,E2 -18082.277} C_VEL
LIN {X 0,Y 261.208,Z 705.476,A -85,B 0,C 180,E1 -18084.573,E2 -18084.573} C_VEL
LIN {X 0,Y 261.131,Z 707.168,A -85,B 0,C 180,E1 -18086.914,E2 -18086.914} C_VEL
LIN {X 0,Y 261.117,Z 707.778,A -85,B 0,C 180,E1 -18088.457,E2 -18088.457} C_VEL
LIN {X 0,Y 261.138,Z 707.993,A -85,B 0,C 180,E1 -18090,E2 -18090} C_VEL
LIN {X 0,Y 261.161,Z 707.769,A -85,B 0,C 180,E1 -18091.542,E2 -18091.542} C_VEL
LIN {X 0,Y 261.157,Z 707.154,A -85,B 0,C 180,E1 -18093.085,E2 -18093.085} C_VEL
LIN {X 0,Y 261.23,Z 705.401,A -85,B 0,C 180,E1 -18095.479,E2 -18095.479} C_VEL
LIN {X 0,Y 261.659,Z 701.757,A -85,B 0,C 180,E1 -18098.495,E2 -18098.495} C_VEL
LIN {X 0,Y 262.366,Z 697.732,A -85,B 0,C 180,E1 -18100.807,E2 -18100.807} C_VEL
LIN {X 0,Y 263.516,Z 691.523,A -85,B 0,C 180,E1 -18103.495,E2 -18103.495} C_VEL
LIN {X 0,Y 265.016,Z 684.75,A -85,B 0,C 180,E1 -18105.773,E2 -18105.773} C_VEL
LIN {X 0,Y 266.426,Z 677.814,A -85,B 0,C 180,E1 -18107.659,E2 -18107.659} C_VEL
LIN {X 0,Y 268.281,Z 668.563,A -85,B 0,C 180,E1 -18109.693,E2 -18109.693} C_VEL
LIN {X 0,Y 270.065,Z 659.063,A -85,B 0,C 180,E1 -18111.366,E2 -18111.366} C_VEL
LIN {X 0,Y 271.889,Z 648.792,A -85,B 0,C 180,E1 -18112.813,E2 -18112.813} C_VEL
LIN {X 0,Y 273.606,Z 637.496,A -85,B 0,C 180,E1 -18114.065,E2 -18114.065} C_VEL
LIN {X 0,Y 274.353,Z 631.714,A -85,B 0,C 180,E1 -18114.599,E2 -18114.599} C_VEL
LIN {X 0,Y 278.752,Z 620.551,A -85,B 0,C 180,E1 -18116.585,E2 -18116.585} C_VEL
LIN {X 0,Y 283.333,Z 608.156,A -85,B 0,C 180,E1 -18118.32,E2 -18118.32} C_VEL
LIN {X 0,Y 287.929,Z 594.272,A -85,B 0,C 180,E1 -18119.823,E2 -18119.823} C_VEL
LIN {X 0,Y 291.797,Z 580.429,A -85,B 0,C 180,E1 -18120.986,E2 -18120.986} C_VEL
LIN {X 0,Y 295.098,Z 566.362,A -85,B 0,C 180,E1 -18121.898,E2 -18121.898} C_VEL
LIN {X 0,Y 297.98,Z 549.804,A -85,B 0,C 180,E1 -18122.701,E2 -18122.701} C_VEL
LIN {X 0,Y 300.021,Z 534.263,A -85,B 0,C 180,E1 -18123.409,E2 -18123.409} C_VEL
LIN {X 0,Y 301.029,Z 520.837,A -85,B 0,C 180,E1 -18124.302,E2 -18124.302} C_VEL
LIN {X 0,Y 301.513,Z 507.186,A -85,B 0,C 180,E1 -18125.475,E2 -18125.475} C_VEL
LIN {X 0,Y 301.679,Z 492.517,A -85,B 0,C 180,E1 -18127.048,E2 -18127.048} C_VEL
LIN {X 0,Y 301.651,Z 484.391,A -85,B 0,C 180,E1 -18128.099,E2 -18128.099} C_VEL
LIN {X 0,Y 299.918,Z 477.405,A -85,B 0,C 180,E1 -18130.193,E2 -18130.193} C_VEL
LIN {X 0,Y 298.392,Z 471.37,A -85,B 0,C 180,E1 -18132.943,E2 -18132.943} C_VEL
LIN {X 0,Y 297.964,Z 468.191,A -85,B 0,C 180,E1 -18135.127,E2 -18135.127} C_VEL
LIN {X 0,Y 298.538,Z 465.913,A -85,B 0,C 180,E1 -18138.04,E2 -18138.04} C_VEL
LIN {X 0,Y 300.165,Z 465.672,A -85,B 0,C 180,E1 -18140.593,E2 -18140.593} C_VEL
LIN {X 0,Y 302.163,Z 466.637,A -85,B 0,C 180,E1 -18142.576,E2 -18142.576} C_VEL
LIN {X 0,Y 304.545,Z 468.885,A -85,B 0,C 180,E1 -18144.429,E2 -18144.429} C_VEL
LIN {X 0,Y 306.868,Z 471.66,A -85,B 0,C 180,E1 -18145.901,E2 -18145.901} C_VEL
LIN {X 0,Y 307.681,Z 473.675,A -85,B 0,C 180,E1 -18146.504,E2 -18146.504} C_VEL
LIN {X 0,Y 302.786,Z 506.645,A -85,B 0,C 180,E1 -18148.077,E2 -18148.077} C_VEL
LIN {X 0,Y 300.971,Z 521.165,A -85,B 0,C 180,E1 -18148.941,E2 -18148.941} C_VEL
LIN {X 0,Y 299.035,Z 533.112,A -85,B 0,C 180,E1 -18149.844,E2 -18149.844} C_VEL
LIN {X 0,Y 296.593,Z 544.462,A -85,B 0,C 180,E1 -18150.937,E2 -18150.937} C_VEL
LIN {X 0,Y 293.292,Z 557.093,A -85,B 0,C 180,E1 -18152.492,E2 -18152.492} C_VEL
LIN {X 0,Y 289.862,Z 567.743,A -85,B 0,C 180,E1 -18154.124,E2 -18154.124} C_VEL
LIN {X 0,Y 286.767,Z 576.146,A -85,B 0,C 180,E1 -18155.764,E2 -18155.764} C_VEL
LIN {X 0,Y 283.275,Z 584.524,A -85,B 0,C 180,E1 -18157.768,E2 -18157.768} C_VEL
LIN {X 0,Y 280.515,Z 590.229,A -85,B 0,C 180,E1 -18159.466,E2 -18159.466} C_VEL
LIN {X 0,Y 277.444,Z 595.829,A -85,B 0,C 180,E1 -18161.54,E2 -18161.54} C_VEL
LIN {X 0,Y 274.685,Z 600.222,A -85,B 0,C 180,E1 -18163.654,E2 -18163.654} C_VEL
LIN {X 0,Y 272.95,Z 602.516,A -85,B 0,C 180,E1 -18165.079,E2 -18165.079} C_VEL
LIN {X 0,Y 270.063,Z 605.705,A -85,B 0,C 180,E1 -18167.984,E2 -18167.984} C_VEL
LIN {X 0,Y 268.731,Z 606.666,A -85,B 0,C 180,E1 -18169.452,E2 -18169.452} C_VEL
LIN {X 0,Y 267.542,Z 607.183,A -85,B 0,C 180,E1 -18170.932,E2 -18170.932} C_VEL
LIN {X 0,Y 266.594,Z 607.27,A -85,B 0,C 180,E1 -18172.426,E2 -18172.426} C_VEL
LIN {X 0,Y 265.873,Z 606.929,A -85,B 0,C 180,E1 -18173.931,E2 -18173.931} C_VEL
LIN {X 0,Y 265.266,Z 606.14,A -85,B 0,C 180,E1 -18175.441,E2 -18175.441} C_VEL
LIN {X 0,Y 264.567,Z 604.968,A -85,B 0,C 180,E1 -18176.955,E2 -18176.955} C_VEL
LIN {X 0,Y 263.805,Z 602.392,A -85,B 0,C 180,E1 -18179.237,E2 -18179.237} C_VEL
LIN {X 0,Y 263.419,Z 598.788,A -85,B 0,C 180,E1 -18181.529,E2 -18181.529} C_VEL
LIN {X 0,Y 263.237,Z 594.095,A -85,B 0,C 180,E1 -18183.827,E2 -18183.827} C_VEL
LIN {X 0,Y 263.325,Z 588.168,A -85,B 0,C 180,E1 -18186.129,E2 -18186.129} C_VEL
LIN {X 0,Y 263.734,Z 580.807,A -85,B 0,C 180,E1 -18188.428,E2 -18188.428} C_VEL
LIN {X 0,Y 264.238,Z 571.744,A -85,B 0,C 180,E1 -18190.73,E2 -18190.73} C_VEL
